LIN {X 0,Y 185.517,Z 546.376,A -85,B 0,C 180,E1 -22264.627,E2 -22264.627} C_VEL
LIN {X 0,Y 185.564,Z 546.364,A -85,B 0,C 180,E1 -22267.314,E2 -22267.314} C_VEL
LIN {X 0,Y 185.581,Z 546.361,A -85,B 0,C 180,E1 -22270.766,E2 -22270.766} C_VEL
LIN {X 0,Y 185.578,Z 546.362,A -85,B 0,C 180,E1 -22276.016,E2 -22276.016} C_VEL
LIN {X 0,Y 185.556,Z 546.364,A -85,B 0,C 180,E1 -22279.92,E2 -22279.92} C_VEL
LIN {X 0,Y 185.571,Z 546.368,A -85,B 0,C 180,E1 -22282.704,E2 -22282.704} C_VEL
LIN {X 0,Y 185.54,Z 546.354,A -85,B 0,C 180,E1 -22287.976,E2 -22287.976} C_VEL
LIN {X 0,Y 185.578,Z 546.361,A -85,B 0,C 180,E1 -22290.576,E2 -22290.576} C_VEL
LIN {X 0,Y 185.575,Z 546.366,A -85,B 0,C 180,E1 -22295.382,E2 -22295.382} C_VEL
LIN {X 0,Y 185.668,Z 546.345,A -85,B 0,C 180,E1 -22301.136,E2 -22301.136} C_VEL
LIN {X 0,Y 185.689,Z 546.352,A -85,B 0,C 180,E1 -22304.638,E2 -22304.638} C_VEL
LIN {X 0,Y 185.92,Z 546.306,A -85,B 0,C 180,E1 -22309.36,E2 -22309.36} C_VEL
LIN {X 0,Y 185.958,Z 546.315,A -85,B 0,C 180,E1 -22313.491,E2 -22313.491} C_VEL
LIN {X 0,Y 186.204,Z 546.281,A -85,B 0,C 180,E1 -22317.838,E2 -22317.838} C_VEL
LIN {X 0,Y 186.405,Z 546.247,A -85,B 0,C 180,E1 -22320.001,E2 -22320.001} C_VEL
LIN {X 0,Y 185.935,Z 546.319,A -85,B 0,C 180,E1 -22324.337,E2 -22324.337} C_VEL
LIN {X 0,Y 185.984,Z 546.307,A -85,B 0,C 180,E1 -22328.695,E2 -22328.695} C_VEL
LIN {X 0,Y 185.726,Z 546.349,A -85,B 0,C 180,E1 -22333.124,E2 -22333.124} C_VEL
LIN {X 0,Y 185.687,Z 546.346,A -85,B 0,C 180,E1 -22337.626,E2 -22337.626} C_VEL
LIN {X 0,Y 185.595,Z 546.364,A -85,B 0,C 180,E1 -22342.253,E2 -22342.253} C_VEL
LIN {X 0,Y 185.561,Z 546.372,A -85,B 0,C 180,E1 -22347.033,E2 -22347.033} C_VEL
LIN {X 0,Y 185.578,Z 546.364,A -85,B 0,C 180,E1 -22349.494,E2 -22349.494} C_VEL
LIN {X 0,Y 185.518,Z 546.372,A -85,B 0,C 180,E1 -22354.629,E2 -22354.629} C_VEL
LIN {X 0,Y 185.544,Z 546.371,A -85,B 0,C 180,E1 -22357.305,E2 -22357.305} C_VEL
LIN {X 0,Y 185.492,Z 546.377,A -85,B 0,C 180,E1 -22360.734,E2 -22360.734} C_VEL
LIN {X 0,Y 185.569,Z 546.427,A -85,B 0,C 180,E1 -22365.591,E2 -22365.591} C_VEL
LIN {X 0,Y 187.78,Z 555.622,A -85,B 0,C 180,E1 -22370.488,E2 -22370.488} C_VEL
LIN {X 0,Y 187.975,Z 556.393,A -85,B 0,C 180,E1 -22370.714,E2 -22370.714} C_VEL
LIN {X 0,Y 195.844,Z 575.592,A -85,B 0,C 180,E1 -22372.988,E2 -22372.988} C_VEL
LIN {X 0,Y 200.611,Z 588.551,A -85,B 0,C 180,E1 -22374.325,E2 -22374.325} C_VEL
LIN {X 0,Y 203.905,Z 619.674,A -85,B 0,C 180,E1 -22376.185,E2 -22376.185} C_VEL
LIN {X 0,Y 202.479,Z 649.546,A -85,B 0,C 180,E1 -22377.312,E2 -22377.312} C_VEL
LIN {X 0,Y 201.533,Z 655.365,A -85,B 0,C 180,E1 -22377.442,E2 -22377.442} C_VEL
LIN {X 0,Y 198.317,Z 664.756,A -85,B 0,C 180,E1 -22377.495,E2 -22377.495} C_VEL
LIN {X 0,Y 194.902,Z 674.04,A -85,B 0,C 180,E1 -22377.731,E2 -22377.731} C_VEL
LIN {X 0,Y 193.615,Z 679.689,A -85,B 0,C 180,E1 -22378.095,E2 -22378.095} C_VEL
LIN {X 0,Y 191.784,Z 691.638,A -85,B 0,C 180,E1 -22379.287,E2 -22379.287} C_VEL
LIN {X 0,Y 189.555,Z 703.367,A -85,B 0,C 180,E1 -22380.882,E2 -22380.882} C_VEL
LIN {X 0,Y 186.984,Z 714.728,A -85,B 0,C 180,E1 -22382.889,E2 -22382.889} C_VEL
LIN {X 0,Y 184.523,Z 725.042,A -85,B 0,C 180,E1 -22385.232,E2 -22385.232} C_VEL
LIN {X 0,Y 182.216,Z 734.209,A -85,B 0,C 180,E1 -22387.873,E2 -22387.873} C_VEL
LIN {X 0,Y 180.274,Z 741.969,A -85,B 0,C 180,E1 -22390.648,E2 -22390.648} C_VEL
LIN {X 0,Y 178.473,Z 749.457,A -85,B 0,C 180,E1 -22394,E2 -22394} C_VEL
LIN {X 0,Y 177.209,Z 755.433,A -85,B 0,C 180,E1 -22397.401,E2 -22397.401} C_VEL
LIN {X 0,Y 176.559,Z 760.116,A -85,B 0,C 180,E1 -22400.839,E2 -22400.839} C_VEL
LIN {X 0,Y 176.397,Z 764.143,A -85,B 0,C 180,E1 -22404.915,E2 -22404.915} C_VEL
LIN {X 0,Y 176.439,Z 766.075,A -85,B 0,C 180,E1 -22407.717,E2 -22407.717} C_VEL
LIN {X 0,Y 176.506,Z 767.141,A -85,B 0,C 180,E1 -22410,E2 -22410} C_VEL
LIN {X 0,Y 176.35,Z 767.745,A -85,B 0,C 180,E1 -22412.284,E2 -22412.284} C_VEL
LIN {X 0,Y 176.194,Z 767.759,A -85,B 0,C 180,E1 -22416.873,E2 -22416.873} C_VEL
LIN {X 0,Y 176.425,Z 767.177,A -85,B 0,C 180,E1 -22419.168,E2 -22419.168} C_VEL
LIN {X 0,Y 177.547,Z 764.782,A -85,B 0,C 180,E1 -22423.739,E2 -22423.739} C_VEL
LIN {X 0,Y 179.222,Z 761.932,A -85,B 0,C 180,E1 -22427.103,E2 -22427.103} C_VEL
LIN {X 0,Y 181.458,Z 758.092,A -85,B 0,C 180,E1 -22430.4,E2 -22430.4} C_VEL
LIN {X 0,Y 184.566,Z 752.928,A -85,B 0,C 180,E1 -22433.731,E2 -22433.731} C_VEL
LIN {X 0,Y 188.364,Z 745.947,A -85,B 0,C 180,E1 -22437.197,E2 -22437.197} C_VEL
LIN {X 0,Y 192.524,Z 738.16,A -85,B 0,C 180,E1 -22440.127,E2 -22440.127} C_VEL
LIN {X 0,Y 197.285,Z 728.483,A -85,B 0,C 180,E1 -22442.905,E2 -22442.905} C_VEL
LIN {X 0,Y 201.625,Z 718.591,A -85,B 0,C 180,E1 -22445.108,E2 -22445.108} C_VEL
LIN {X 0,Y 205.882,Z 707.605,A -85,B 0,C 180,E1 -22446.987,E2 -22446.987} C_VEL
LIN {X 0,Y 209.356,Z 697.038,A -85,B 0,C 180,E1 -22448.391,E2 -22448.391} C_VEL
LIN {X 0,Y 212.547,Z 685.576,A -85,B 0,C 180,E1 -22449.531,E2 -22449.531} C_VEL
LIN {X 0,Y 215.285,Z 672.899,A -85,B 0,C 180,E1 -22450.452,E2 -22450.452} C_VEL
LIN {X 0,Y 217.072,Z 659.892,A -85,B 0,C 180,E1 -22451.115,E2 -22451.115} C_VEL
LIN {X 0,Y 219.901,Z 624.876,A -85,B 0,C 180,E1 -22452.357,E2 -22452.357} C_VEL
LIN {X 0,Y 219.369,Z 614.997,A -85,B 0,C 180,E1 -22453.156,E2 -22453.156} C_VEL
LIN {X 0,Y 215.934,Z 605.716,A -85,B 0,C 180,E1 -22455.054,E2 -22455.054} C_VEL
LIN {X 0,Y 212.067,Z 596.949,A -85,B 0,C 180,E1 -22457.291,E2 -22457.291} C_VEL
LIN {X 0,Y 208.689,Z 590.362,A -85,B 0,C 180,E1 -22459.448,E2 -22459.448} C_VEL
LIN {X 0,Y 206.695,Z 586.633,A -85,B 0,C 180,E1 -22460.819,E2 -22460.819} C_VEL
LIN {X 0,Y 204.07,Z 581.906,A -85,B 0,C 180,E1 -22462.843,E2 -22462.843} C_VEL
LIN {X 0,Y 200.633,Z 575.973,A -85,B 0,C 180,E1 -22465.911,E2 -22465.911} C_VEL
LIN {X 0,Y 196.518,Z 569.368,A -85,B 0,C 180,E1 -22470.809,E2 -22470.809} C_VEL
LIN {X 0,Y 193.752,Z 565.553,A -85,B 0,C 180,E1 -22476.225,E2 -22476.225} C_VEL
LIN {X 0,Y 193.121,Z 564.144,A -85,B 0,C 180,E1 -22479.251,E2 -22479.251} C_VEL
LIN {X 0,Y 193.05,Z 563.979,A -85,B 0,C 180,E1 -22483.067,E2 -22483.067} C_VEL
LIN {X 0,Y 195.749,Z 565.397,A -85,B 0,C 180,E1 -22490.374,E2 -22490.374} C_VEL
LIN {X 0,Y 197.208,Z 568.439,A -85,B 0,C 180,E1 -22492.778,E2 -22492.778} C_VEL
LIN {X 0,Y 199.601,Z 570.637,A -85,B 0,C 180,E1 -22495.487,E2 -22495.487} C_VEL
LIN {X 0,Y 200.336,Z 571.297,A -85,B 0,C 180,E1 -22496.201,E2 -22496.201} C_VEL
LIN {X 0,Y 202.709,Z 574.7,A -85,B 0,C 180,E1 -22498.455,E2 -22498.455} C_VEL
LIN {X 0,Y 206.086,Z 579.678,A -85,B 0,C 180,E1 -22501.122,E2 -22501.122} C_VEL
LIN {X 0,Y 210.138,Z 585.674,A -85,B 0,C 180,E1 -22503.834,E2 -22503.834} C_VEL
LIN {X 0,Y 215.436,Z 594.551,A -85,B 0,C 180,E1 -22506.911,E2 -22506.911} C_VEL
LIN {X 0,Y 219.159,Z 601.544,A -85,B 0,C 180,E1 -22508.844,E2 -22508.844} C_VEL
LIN {X 0,Y 221.223,Z 605.714,A -85,B 0,C 180,E1 -22509.853,E2 -22509.853} C_VEL
LIN {X 0,Y 217.676,Z 648.267,A -85,B 0,C 180,E1 -22511.39,E2 -22511.39} C_VEL
LIN {X 0,Y 215.672,Z 661.882,A -85,B 0,C 180,E1 -22512.224,E2 -22512.224} C_VEL
LIN {X 0,Y 213.173,Z 674.111,A -85,B 0,C 180,E1 -22513.342,E2 -22513.342} C_VEL
LIN {X 0,Y 210.175,Z 685.358,A -85,B 0,C 180,E1 -22514.715,E2 -22514.715} C_VEL
LIN {X 0,Y 206.233,Z 697.154,A -85,B 0,C 180,E1 -22516.568,E2 -22516.568} C_VEL
LIN {X 0,Y 202.085,Z 707.52,A -85,B 0,C 180,E1 -22518.702,E2 -22518.702} C_VEL
LIN {X 0,Y 197.666,Z 717.189,A -85,B 0,C 180,E1 -22521.271,E2 -22521.271} C_VEL
LIN {X 0,Y 193.61,Z 724.993,A -85,B 0,C 180,E1 -22523.922,E2 -22523.922} C_VEL
LIN {X 0,Y 189.421,Z 732.125,A -85,B 0,C 180,E1 -22527.071,E2 -22527.071} C_VEL
LIN {X 0,Y 186.39,Z 736.986,A -85,B 0,C 180,E1 -22529.863,E2 -22529.863} C_VEL
LIN {X 0,Y 183.741,Z 740.865,A -85,B 0,C 180,E1 -22532.704,E2 -22532.704} C_VEL
LIN {X 0,Y 180.564,Z 745.035,A -85,B 0,C 180,E1 -22537.071,E2 -22537.071} C_VEL
LIN {X 0,Y 178.287,Z 747.512,A -85,B 0,C 180,E1 -22541.5,E2 -22541.5} C_VEL
LIN {X 0,Y 176.895,Z 748.349,A -85,B 0,C 180,E1 -22545.652,E2 -22545.652} C_VEL
LIN {X 0,Y 176.092,Z 747.755,A -85,B 0,C 180,E1 -22550.315,E2 -22550.315} C_VEL
LIN {X 0,Y 175.986,Z 746.527,A -85,B 0,C 180,E1 -22553.201,E2 -22553.201} C_VEL
LIN {X 0,Y 176.304,Z 744.071,A -85,B 0,C 180,E1 -22556.835,E2 -22556.835} C_VEL
LIN {X 0,Y 177.175,Z 740.148,A -85,B 0,C 180,E1 -22560.769,E2 -22560.769} C_VEL
LIN {X 0,Y 178.282,Z 735.346,A -85,B 0,C 180,E1 -22564.303,E2 -22564.303} C_VEL
LIN {X 0,Y 179.981,Z 728.514,A -85,B 0,C 180,E1 -22568.114,E2 -22568.114} C_VEL
LIN {X 0,Y 181.997,Z 720.884,A -85,B 0,C 180,E1 -22571.423,E2 -22571.423} C_VEL
LIN {X 0,Y 184.362,Z 711.833,A -85,B 0,C 180,E1 -22574.524,E2 -22574.524} C_VEL
LIN {X 0,Y 186.903,Z 701.354,A -85,B 0,C 180,E1 -22577.332,E2 -22577.332} C_VEL
LIN {X 0,Y 189.262,Z 690.78,A -85,B 0,C 180,E1 -22579.571,E2 -22579.571} C_VEL
LIN {X 0,Y 191.53,Z 678.663,A -85,B 0,C 180,E1 -22581.56,E2 -22581.56} C_VEL
LIN {X 0,Y 193.414,Z 666.412,A -85,B 0,C 180,E1 -22583.087,E2 -22583.087} C_VEL
LIN {X 0,Y 194.854,Z 653.682,A -85,B 0,C 180,E1 -22584.243,E2 -22584.243} C_VEL
LIN {X 0,Y 195.962,Z 639.684,A -85,B 0,C 180,E1 -22585.049,E2 -22585.049} C_VEL
LIN {X 0,Y 198.703,Z 589.027,A -85,B 0,C 180,E1 -22586.989,E2 -22586.989} C_VEL
LIN {X 0,Y 192.071,Z 573.5,A -85,B 0,C 180,E1 -22588.782,E2 -22588.782} C_VEL
LIN {X 0,Y 182.607,Z 554.067,A -85,B 0,C 180,E1 -22591.435,E2 -22591.435} C_VEL
LIN {X 0,Y 180.336,Z 550.24,A -85,B 0,C 180,E1 -22592.077,E2 -22592.077} C_VEL
LIN {X 0,Y 179.153,Z 547.494,A -85,B 0,C 180,E1 -22592.459,E2 -22592.459} C_VEL
LIN {X 0,Y 179.086,Z 547.178,A -85,B 0,C 180,E1 -22592.53,E2 -22592.53} C_VEL
LIN {X 0,Y 178.976,Z 547.189,A -85,B 0,C 180,E1 -22599.037,E2 -22599.037} C_VEL
LIN {X 0,Y 178.685,Z 547.223,A -85,B 0,C 180,E1 -22603.65,E2 -22603.65} C_VEL
LIN {X 0,Y 178.647,Z 547.229,A -85,B 0,C 180,E1 -22608.344,E2 -22608.344} C_VEL
LIN {X 0,Y 178.508,Z 547.247,A -85,B 0,C 180,E1 -22613.185,E2 -22613.185} C_VEL
LIN {X 0,Y 178.484,Z 547.251,A -85,B 0,C 180,E1 -22618.197,E2 -22618.197} C_VEL
LIN {X 0,Y 178.476,Z 547.253,A -85,B 0,C 180,E1 -22620.791,E2 -22620.791} C_VEL
LIN {X 0,Y 178.481,Z 547.251,A -85,B 0,C 180,E1 -22624.22,E2 -22624.22} C_VEL
LIN {X 0,Y 178.482,Z 547.241,A -85,B 0,C 180,E1 -22629.051,E2 -22629.051} C_VEL
LIN {X 0,Y 178.513,Z 547.246,A -85,B 0,C 180,E1 -22632.011,E2 -22632.011} C_VEL
LIN {X 0,Y 178.525,Z 547.243,A -85,B 0,C 180,E1 -22635.12,E2 -22635.12} C_VEL
LIN {X 0,Y 178.508,Z 547.232,A -85,B 0,C 180,E1 -22638.42,E2 -22638.42} C_VEL
LIN {X 0,Y 178.484,Z 547.249,A -85,B 0,C 180,E1 -22643.799,E2 -22643.799} C_VEL
LIN {X 0,Y 178.487,Z 547.24,A -85,B 0,C 180,E1 -22646.548,E2 -22646.548} C_VEL
LIN {X 0,Y 178.518,Z 547.239,A -85,B 0,C 180,E1 -22650.007,E2 -22650.007} C_VEL
LIN {X 0,Y 178.515,Z 547.248,A -85,B 0,C 180,E1 -22654.886,E2 -22654.886} C_VEL
LIN {X 0,Y 178.616,Z 547.221,A -85,B 0,C 180,E1 -22660.787,E2 -22660.787} C_VEL
LIN {X 0,Y 178.656,Z 547.227,A -85,B 0,C 180,E1 -22666.349,E2 -22666.349} C_VEL
LIN {X 0,Y 178.934,Z 547.174,A -85,B 0,C 180,E1 -22670.962,E2 -22670.962} C_VEL
LIN {X 0,Y 179.15,Z 547.16,A -85,B 0,C 180,E1 -22677.753,E2 -22677.753} C_VEL
LIN {X 0,Y 179.368,Z 547.123,A -85,B 0,C 180,E1 -22680.001,E2 -22680.001} C_VEL
LIN {X 0,Y 178.882,Z 547.198,A -85,B 0,C 180,E1 -22684.508,E2 -22684.508} C_VEL
LIN {X 0,Y 178.911,Z 547.186,A -85,B 0,C 180,E1 -22689.041,E2 -22689.041} C_VEL
LIN {X 0,Y 178.654,Z 547.23,A -85,B 0,C 180,E1 -22693.654,E2 -22693.654} C_VEL
LIN {X 0,Y 178.621,Z 547.231,A -85,B 0,C 180,E1 -22699.217,E2 -22699.217} C_VEL
LIN {X 0,Y 178.523,Z 547.242,A -85,B 0,C 180,E1 -22705.119,E2 -22705.119} C_VEL
LIN {X 0,Y 178.522,Z 547.243,A -85,B 0,C 180,E1 -22709.995,E2 -22709.995} C_VEL
LIN {X 0,Y 178.495,Z 547.247,A -85,B 0,C 180,E1 -22714.226,E2 -22714.226} C_VEL
LIN {X 0,Y 178.421,Z 547.262,A -85,B 0,C 180,E1 -22719.069,E2 -22719.069} C_VEL
LIN {X 0,Y 178.493,Z 547.298,A -85,B 0,C 180,E1 -22724.67,E2 -22724.67} C_VEL
LIN {X 0,Y 180.414,Z 555.176,A -85,B 0,C 180,E1 -22729.08,E2 -22729.08} C_VEL
LIN {X 0,Y 180.613,Z 555.846,A -85,B 0,C 180,E1 -22729.316,E2 -22729.316} C_VEL
LIN {X 0,Y 188.551,Z 574.701,A -85,B 0,C 180,E1 -22731.729,E2 -22731.729} C_VEL
LIN {X 0,Y 194.574,Z 591.255,A -85,B 0,C 180,E1 -22733.529,E2 -22733.529} C_VEL
LIN {X 0,Y 197.522,Z 620.88,A -85,B 0,C 180,E1 -22735.353,E2 -22735.353} C_VEL
LIN {X 0,Y 195.045,Z 666.296,A -85,B 0,C 180,E1 -22737.172,E2 -22737.172} C_VEL
LIN {X 0,Y 193.812,Z 678.176,A -85,B 0,C 180,E1 -22737.973,E2 -22737.973} C_VEL
LIN {X 0,Y 193.615,Z 679.689,A -85,B 0,C 180,E1 -22738.095,E2 -22738.095} C_VEL
LIN {X 0,Y 192.148,Z 685.25,A -85,B 0,C 180,E1 -22738.513,E2 -22738.513} C_VEL
LIN {X 0,Y 187.941,Z 694.002,A -85,B 0,C 180,E1 -22739.154,E2 -22739.154} C_VEL
LIN {X 0,Y 183.605,Z 702.435,A -85,B 0,C 180,E1 -22740.042,E2 -22740.042} C_VEL
LIN {X 0,Y 181.958,Z 707.489,A -85,B 0,C 180,E1 -22740.843,E2 -22740.843} C_VEL
LIN {X 0,Y 179.215,Z 719.04,A -85,B 0,C 180,E1 -22743.194,E2 -22743.194} C_VEL
LIN {X 0,Y 177.031,Z 727.49,A -85,B 0,C 180,E1 -22745.365,E2 -22745.365} C_VEL
LIN {X 0,Y 174.552,Z 736.495,A -85,B 0,C 180,E1 -22748.221,E2 -22748.221} C_VEL
LIN {X 0,Y 172.508,Z 744.812,A -85,B 0,C 180,E1 -22751.595,E2 -22751.595} C_VEL
LIN {X 0,Y 170.822,Z 751.631,A -85,B 0,C 180,E1 -22755.1,E2 -22755.1} C_VEL
LIN {X 0,Y 169.697,Z 757.854,A -85,B 0,C 180,E1 -22759.259,E2 -22759.259} C_VEL
LIN {X 0,Y 169.31,Z 761.846,A -85,B 0,C 180,E1 -22762.847,E2 -22762.847} C_VEL
LIN {X 0,Y 169.328,Z 763.874,A -85,B 0,C 180,E1 -22765.238,E2 -22765.238} C_VEL
LIN {X 0,Y 169.355,Z 765.452,A -85,B 0,C 180,E1 -22767.622,E2 -22767.622} C_VEL
LIN {X 0,Y 169.44,Z 766.598,A -85,B 0,C 180,E1 -22770,E2 -22770} C_VEL
LIN {X 0,Y 169.114,Z 767.495,A -85,B 0,C 180,E1 -22774.131,E2 -22774.131} C_VEL
LIN {X 0,Y 169.126,Z 767.366,A -85,B 0,C 180,E1 -22777.161,E2 -22777.161} C_VEL
LIN {X 0,Y 169.379,Z 766.846,A -85,B 0,C 180,E1 -22779.553,E2 -22779.553} C_VEL
LIN {X 0,Y 169.863,Z 765.923,A -85,B 0,C 180,E1 -22781.939,E2 -22781.939} C_VEL
LIN {X 0,Y 171.721,Z 762.851,A -85,B 0,C 180,E1 -22786.647,E2 -22786.647} C_VEL
LIN {X 0,Y 173.974,Z 759.469,A -85,B 0,C 180,E1 -22790.082,E2 -22790.082} C_VEL
LIN {X 0,Y 176.85,Z 755.059,A -85,B 0,C 180,E1 -22793.415,E2 -22793.415} C_VEL
LIN {X 0,Y 180.784,Z 748.483,A -85,B 0,C 180,E1 -22797.179,E2 -22797.179} C_VEL
LIN {X 0,Y 184.954,Z 741.38,A -85,B 0,C 180,E1 -22800.23,E2 -22800.23} C_VEL
LIN {X 0,Y 189.674,Z 732.613,A -85,B 0,C 180,E1 -22803.129,E2 -22803.129} C_VEL
LIN {X 0,Y 194.104,Z 723.731,A -85,B 0,C 180,E1 -22805.402,E2 -22805.402} C_VEL
LIN {X 0,Y 198.793,Z 712.911,A -85,B 0,C 180,E1 -22807.577,E2 -22807.577} C_VEL
LIN {X 0,Y 202.843,Z 702.103,A -85,B 0,C 180,E1 -22809.22,E2 -22809.22} C_VEL
LIN {X 0,Y 206.595,Z 690.184,A -85,B 0,C 180,E1 -22810.585,E2 -22810.585} C_VEL
LIN {X 0,Y 209.73,Z 677.93,A -85,B 0,C 180,E1 -22811.598,E2 -22811.598} C_VEL
LIN {X 0,Y 212.106,Z 664.304,A -85,B 0,C 180,E1 -22812.4,E2 -22812.4} C_VEL
LIN {X 0,Y 214.091,Z 644.025,A -85,B 0,C 180,E1 -22813.158,E2 -22813.158} C_VEL
LIN {X 0,Y 215.57,Z 625.879,A -85,B 0,C 180,E1 -22813.819,E2 -22813.819} C_VEL
LIN {X 0,Y 215.277,Z 618.3,A -85,B 0,C 180,E1 -22814.445,E2 -22814.445} C_VEL
LIN {X 0,Y 211.9,Z 609.02,A -85,B 0,C 180,E1 -22816.466,E2 -22816.466} C_VEL
LIN {X 0,Y 208.766,Z 601.726,A -85,B 0,C 180,E1 -22818.464,E2 -22818.464} C_VEL
LIN {X 0,Y 205.691,Z 595.44,A -85,B 0,C 180,E1 -22820.575,E2 -22820.575} C_VEL
LIN {X 0,Y 203.613,Z 591.42,A -85,B 0,C 180,E1 -22822.167,E2 -22822.167} C_VEL
LIN {X 0,Y 201.707,Z 587.854,A -85,B 0,C 180,E1 -22823.759,E2 -22823.759} C_VEL
LIN {X 0,Y 198.706,Z 582.299,A -85,B 0,C 180,E1 -22826.677,E2 -22826.677} C_VEL
LIN {X 0,Y 195.087,Z 576.109,A -85,B 0,C 180,E1 -22831.317,E2 -22831.317} C_VEL
LIN {X 0,Y 192.499,Z 572.282,A -85,B 0,C 180,E1 -22836.89,E2 -22836.89} C_VEL
LIN {X 0,Y 192.023,Z 571.108,A -85,B 0,C 180,E1 -22839.722,E2 -22839.722} C_VEL
LIN {X 0,Y 192.16,Z 571.117,A -85,B 0,C 180,E1 -22844.079,E2 -22844.079} C_VEL
LIN {X 0,Y 194.484,Z 572.512,A -85,B 0,C 180,E1 -22850.099,E2 -22850.099} C_VEL
LIN {X 0,Y 196.01,Z 575.569,A -85,B 0,C 180,E1 -22852.652,E2 -22852.652} C_VEL
LIN {X 0,Y 198.624,Z 577.973,A -85,B 0,C 180,E1 -22855.631,E2 -22855.631} C_VEL
LIN {X 0,Y 201.392,Z 582.172,A -85,B 0,C 180,E1 -22858.366,E2 -22858.366} C_VEL
LIN {X 0,Y 204.038,Z 586.131,A -85,B 0,C 180,E1 -22860.514,E2 -22860.514} C_VEL
LIN {X 0,Y 207.661,Z 591.827,A -85,B 0,C 180,E1 -22863.105,E2 -22863.105} C_VEL
LIN {X 0,Y 212.638,Z 600.542,A -85,B 0,C 180,E1 -22866.18,E2 -22866.18} C_VEL
LIN {X 0,Y 216.291,Z 607.643,A -85,B 0,C 180,E1 -22868.166,E2 -22868.166} C_VEL
LIN {X 0,Y 216.856,Z 608.973,A -85,B 0,C 180,E1 -22868.474,E2 -22868.474} C_VEL
LIN {X 0,Y 213.287,Z 648.802,A -85,B 0,C 180,E1 -22869.918,E2 -22869.918} C_VEL
LIN {X 0,Y 211.178,Z 662.261,A -85,B 0,C 180,E1 -22870.741,E2 -22870.741} C_VEL
LIN {X 0,Y 208.758,Z 673.849,A -85,B 0,C 180,E1 -22871.804,E2 -22871.804} C_VEL
LIN {X 0,Y 205.462,Z 685.712,A -85,B 0,C 180,E1 -22873.243,E2 -22873.243} C_VEL
LIN {X 0,Y 201.804,Z 696.255,A -85,B 0,C 180,E1 -22874.882,E2 -22874.882} C_VEL
LIN {X 0,Y 197.506,Z 706.815,A -85,B 0,C 180,E1 -22877.004,E2 -22877.004} C_VEL
LIN {X 0,Y 192.914,Z 716.379,A -85,B 0,C 180,E1 -22879.504,E2 -22879.504} C_VEL
LIN {X 0,Y 188.173,Z 725.092,A -85,B 0,C 180,E1 -22882.463,E2 -22882.463} C_VEL
LIN {X 0,Y 183.333,Z 732.845,A -85,B 0,C 180,E1 -22885.959,E2 -22885.959} C_VEL
LIN {X 0,Y 179.994,Z 737.794,A -85,B 0,C 180,E1 -22888.919,E2 -22888.919} C_VEL
LIN {X 0,Y 176.169,Z 742.919,A -85,B 0,C 180,E1 -22893.098,E2 -22893.098} C_VEL
LIN {X 0,Y 173.118,Z 746.408,A -85,B 0,C 180,E1 -22897.512,E2 -22897.512} C_VEL
LIN {X 0,Y 170.85,Z 748.399,A -85,B 0,C 180,E1 -22902.233,E2 -22902.233} C_VEL
LIN {X 0,Y 169.894,Z 748.785,A -85,B 0,C 180,E1 -22905.314,E2 -22905.314} C_VEL
LIN {X 0,Y 169.252,Z 748.551,A -85,B 0,C 180,E1 -22908.366,E2 -22908.366} C_VEL
LIN {X 0,Y 168.89,Z 747.283,A -85,B 0,C 180,E1 -22912.244,E2 -22912.244} C_VEL
LIN {X 0,Y 169.106,Z 744.855,A -85,B 0,C 180,E1 -22916.219,E2 -22916.219} C_VEL
LIN {X 0,Y 169.946,Z 741.111,A -85,B 0,C 180,E1 -22920.276,E2 -22920.276} C_VEL
LIN {X 0,Y 171.241,Z 735.638,A -85,B 0,C 180,E1 -22924.541,E2 -22924.541} C_VEL
LIN {X 0,Y 173.034,Z 728.659,A -85,B 0,C 180,E1 -22928.559,E2 -22928.559} C_VEL
LIN {X 0,Y 175.02,Z 721.458,A -85,B 0,C 180,E1 -22931.798,E2 -22931.798} C_VEL
LIN {X 0,Y 177.5,Z 712.235,A -85,B 0,C 180,E1 -22935.087,E2 -22935.087} C_VEL
LIN {X 0,Y 180.135,Z 701.766,A -85,B 0,C 180,E1 -22937.993,E2 -22937.993} C_VEL
LIN {X 0,Y 182.583,Z 691.199,A -85,B 0,C 180,E1 -22940.305,E2 -22940.305} C_VEL
LIN {X 0,Y 184.939,Z 679.122,A -85,B 0,C 180,E1 -22942.353,E2 -22942.353} C_VEL
LIN {X 0,Y 186.915,Z 666.847,A -85,B 0,C 180,E1 -22943.93,E2 -22943.93} C_VEL
LIN {X 0,Y 188.406,Z 654.178,A -85,B 0,C 180,E1 -22945.119,E2 -22945.119} C_VEL
LIN {X 0,Y 189.579,Z 639.972,A -85,B 0,C 180,E1 -22945.962,E2 -22945.962} C_VEL
LIN {X 0,Y 192.341,Z 590.76,A -85,B 0,C 180,E1 -22947.906,E2 -22947.906} C_VEL
LIN {X 0,Y 186.259,Z 576.62,A -85,B 0,C 180,E1 -22949.607,E2 -22949.607} C_VEL
LIN {X 0,Y 177.456,Z 558.29,A -85,B 0,C 180,E1 -22952.217,E2 -22952.217} C_VEL
LIN {X 0,Y 173.599,Z 551.821,A -85,B 0,C 180,E1 -22953.361,E2 -22953.361} C_VEL
LIN {X 0,Y 172.119,Z 549.158,A -85,B 0,C 180,E1 -22953.826,E2 -22953.826} C_VEL
LIN {X 0,Y 171.865,Z 548.078,A -85,B 0,C 180,E1 -22954.03,E2 -22954.03} C_VEL
LIN {X 0,Y 171.908,Z 548.07,A -85,B 0,C 180,E1 -22959.412,E2 -22959.412} C_VEL
LIN {X 0,Y 171.607,Z 548.104,A -85,B 0,C 180,E1 -22964.224,E2 -22964.224} C_VEL
LIN {X 0,Y 171.541,Z 548.112,A -85,B 0,C 180,E1 -22969.562,E2 -22969.562} C_VEL
LIN {X 0,Y 171.466,Z 548.122,A -85,B 0,C 180,E1 -22975.616,E2 -22975.616} C_VEL
LIN {X 0,Y 171.438,Z 548.128,A -85,B 0,C 180,E1 -22980.587,E2 -22980.587} C_VEL
LIN {X 0,Y 171.436,Z 548.132,A -85,B 0,C 180,E1 -22985.024,E2 -22985.024} C_VEL
LIN {X 0,Y 171.435,Z 548.118,A -85,B 0,C 180,E1 -22988.841,E2 -22988.841} C_VEL
LIN {X 0,Y 171.449,Z 548.127,A -85,B 0,C 180,E1 -22994.174,E2 -22994.174} C_VEL
LIN {X 0,Y 171.425,Z 548.116,A -85,B 0,C 180,E1 -22999.009,E2 -22999.009} C_VEL
LIN {X 0,Y 171.438,Z 548.127,A -85,B 0,C 180,E1 -23002.056,E2 -23002.056} C_VEL
LIN {X 0,Y 171.412,Z 548.127,A -85,B 0,C 180,E1 -23005.084,E2 -23005.084} C_VEL
LIN {X 0,Y 171.444,Z 548.12,A -85,B 0,C 180,E1 -23010.535,E2 -23010.535} C_VEL
LIN {X 0,Y 171.44,Z 548.125,A -85,B 0,C 180,E1 -23015.8,E2 -23015.8} C_VEL
LIN {X 0,Y 171.572,Z 548.098,A -85,B 0,C 180,E1 -23020.872,E2 -23020.872} C_VEL
LIN {X 0,Y 171.573,Z 548.11,A -85,B 0,C 180,E1 -23025.774,E2 -23025.774} C_VEL
LIN {X 0,Y 171.869,Z 548.052,A -85,B 0,C 180,E1 -23030.587,E2 -23030.587} C_VEL
LIN {X 0,Y 171.82,Z 548.079,A -85,B 0,C 180,E1 -23035.309,E2 -23035.309} C_VEL
LIN {X 0,Y 172.331,Z 547.999,A -85,B 0,C 180,E1 -23040.001,E2 -23040.001} C_VEL
LIN {X 0,Y 171.829,Z 548.077,A -85,B 0,C 180,E1 -23044.693,E2 -23044.693} C_VEL
LIN {X 0,Y 171.847,Z 548.064,A -85,B 0,C 180,E1 -23049.416,E2 -23049.416} C_VEL
LIN {X 0,Y 171.573,Z 548.111,A -85,B 0,C 180,E1 -23054.229,E2 -23054.229} C_VEL
LIN {X 0,Y 171.543,Z 548.115,A -85,B 0,C 180,E1 -23059.563,E2 -23059.563} C_VEL
LIN {X 0,Y 171.461,Z 548.125,A -85,B 0,C 180,E1 -23065.613,E2 -23065.613} C_VEL
LIN {X 0,Y 171.441,Z 548.127,A -85,B 0,C 180,E1 -23070.588,E2 -23070.588} C_VEL
LIN {X 0,Y 171.406,Z 548.132,A -85,B 0,C 180,E1 -23075.033,E2 -23075.033} C_VEL
LIN {X 0,Y 171.382,Z 548.138,A -85,B 0,C 180,E1 -23078.819,E2 -23078.819} C_VEL
LIN {X 0,Y 171.433,Z 548.18,A -85,B 0,C 180,E1 -23083.686,E2 -23083.686} C_VEL
LIN {X 0,Y 173.204,Z 555.248,A -85,B 0,C 180,E1 -23087.799,E2 -23087.799} C_VEL
LIN {X 0,Y 180.811,Z 572.906,A -85,B 0,C 180,E1 -23090.255,E2 -23090.255} C_VEL
LIN {X 0,Y 187.846,Z 591.474,A -85,B 0,C 180,E1 -23092.44,E2 -23092.44} C_VEL
LIN {X 0,Y 188.569,Z 594.359,A -85,B 0,C 180,E1 -23092.703,E2 -23092.703} C_VEL
LIN {X 0,Y 191.147,Z 620.798,A -85,B 0,C 180,E1 -23094.401,E2 -23094.401} C_VEL
LIN {X 0,Y 188.626,Z 665.85,A -85,B 0,C 180,E1 -23096.263,E2 -23096.263} C_VEL
LIN {X 0,Y 187.303,Z 678.136,A -85,B 0,C 180,E1 -23097.12,E2 -23097.12} C_VEL
LIN {X 0,Y 185.289,Z 690.967,A -85,B 0,C 180,E1 -23098.406,E2 -23098.406} C_VEL
LIN {X 0,Y 182.988,Z 702.761,A -85,B 0,C 180,E1 -23100.048,E2 -23100.048} C_VEL
LIN {X 0,Y 181.958,Z 707.489,A -85,B 0,C 180,E1 -23100.843,E2 -23100.843} C_VEL
LIN {X 0,Y 180.251,Z 712.513,A -85,B 0,C 180,E1 -23101.73,E2 -23101.73} C_VEL
LIN {X 0,Y 175.559,Z 720.135,A -85,B 0,C 180,E1 -23103.141,E2 -23103.141} C_VEL
LIN {X 0,Y 170.831,Z 727.218,A -85,B 0,C 180,E1 -23104.802,E2 -23104.802} C_VEL
LIN {X 0,Y 169.094,Z 731.386,A -85,B 0,C 180,E1 -23106.052,E2 -23106.052} C_VEL
LIN {X 0,Y 166.834,Z 739.508,A -85,B 0,C 180,E1 -23109.019,E2 -23109.019} C_VEL
LIN {X 0,Y 164.827,Z 747.311,A -85,B 0,C 180,E1 -23112.635,E2 -23112.635} C_VEL
LIN {X 0,Y 163.282,Z 753.526,A -85,B 0,C 180,E1 -23116.307,E2 -23116.307} C_VEL
LIN {X 0,Y 162.506,Z 758.444,A -85,B 0,C 180,E1 -23120.039,E2 -23120.039} C_VEL
LIN {X 0,Y 162.22,Z 762.173,A -85,B 0,C 180,E1 -23123.782,E2 -23123.782} C_VEL
LIN {X 0,Y 162.273,Z 764.815,A -85,B 0,C 180,E1 -23127.518,E2 -23127.518} C_VEL
LIN {X 0,Y 162.374,Z 766.015,A -85,B 0,C 180,E1 -23130,E2 -23130} C_VEL
LIN {X 0,Y 162.056,Z 766.997,A -85,B 0,C 180,E1 -23134.071,E2 -23134.071} C_VEL
LIN {X 0,Y 162.064,Z 766.973,A -85,B 0,C 180,E1 -23137.475,E2 -23137.475} C_VEL
LIN {X 0,Y 162.874,Z 765.654,A -85,B 0,C 180,E1 -23142.459,E2 -23142.459} C_VEL
LIN {X 0,Y 163.698,Z 764.401,A -85,B 0,C 180,E1 -23144.927,E2 -23144.927} C_VEL
LIN {X 0,Y 166.453,Z 760.658,A -85,B 0,C 180,E1 -23149.741,E2 -23149.741} C_VEL
LIN {X 0,Y 169.249,Z 756.713,A -85,B 0,C 180,E1 -23153.233,E2 -23153.233} C_VEL
LIN {X 0,Y 172.583,Z 751.692,A -85,B 0,C 180,E1 -23156.611,E2 -23156.611} C_VEL
LIN {X 0,Y 176.6,Z 745.48,A -85,B 0,C 180,E1 -23159.831,E2 -23159.831} C_VEL
LIN {X 0,Y 181.293,Z 737.837,A -85,B 0,C 180,E1 -23162.868,E2 -23162.868} C_VEL
LIN {X 0,Y 185.622,Z 730.101,A -85,B 0,C 180,E1 -23165.267,E2 -23165.267} C_VEL
LIN {X 0,Y 190.774,Z 719.712,A -85,B 0,C 180,E1 -23167.766,E2 -23167.766} C_VEL
LIN {X 0,Y 195.396,Z 709.23,A -85,B 0,C 180,E1 -23169.674,E2 -23169.674} C_VEL
LIN {X 0,Y 199.675,Z 697.747,A -85,B 0,C 180,E1 -23171.295,E2 -23171.295} C_VEL
LIN {X 0,Y 203.406,Z 685.688,A -85,B 0,C 180,E1 -23172.524,E2 -23172.524} C_VEL
LIN {X 0,Y 206.535,Z 672.446,A -85,B 0,C 180,E1 -23173.503,E2 -23173.503} C_VEL
LIN {X 0,Y 208.47,Z 659.988,A -85,B 0,C 180,E1 -23174.16,E2 -23174.16} C_VEL
LIN {X 0,Y 211.453,Z 626.855,A -85,B 0,C 180,E1 -23175.361,E2 -23175.361} C_VEL
LIN {X 0,Y 211.246,Z 621.418,A -85,B 0,C 180,E1 -23175.838,E2 -23175.838} C_VEL
LIN {X 0,Y 207.858,Z 611.861,A -85,B 0,C 180,E1 -23178.078,E2 -23178.078} C_VEL
LIN {X 0,Y 204.384,Z 603.729,A -85,B 0,C 180,E1 -23180.541,E2 -23180.541} C_VEL
LIN {X 0,Y 201.594,Z 597.976,A -85,B 0,C 180,E1 -23182.768,E2 -23182.768} C_VEL
LIN {X 0,Y 199.529,Z 593.959,A -85,B 0,C 180,E1 -23184.585,E2 -23184.585} C_VEL
LIN {X 0,Y 196.777,Z 588.577,A -85,B 0,C 180,E1 -23187.498,E2 -23187.498} C_VEL
LIN {X 0,Y 193.654,Z 582.822,A -85,B 0,C 180,E1 -23191.848,E2 -23191.848} C_VEL
LIN {X 0,Y 191.272,Z 578.98,A -85,B 0,C 180,E1 -23197.59,E2 -23197.59} C_VEL
LIN {X 0,Y 190.992,Z 578.159,A -85,B 0,C 180,E1 -23199.608,E2 -23199.608} C_VEL
LIN {X 0,Y 191.102,Z 578.113,A -85,B 0,C 180,E1 -23203.988,E2 -23203.988} C_VEL
LIN {X 0,Y 193.154,Z 579.37,A -85,B 0,C 180,E1 -23209.618,E2 -23209.618} C_VEL
LIN {X 0,Y 194.876,Z 582.735,A -85,B 0,C 180,E1 -23212.609,E2 -23212.609} C_VEL
LIN {X 0,Y 196.996,Z 584.759,A -85,B 0,C 180,E1 -23215.128,E2 -23215.128} C_VEL
LIN {X 0,Y 199.508,Z 588.702,A -85,B 0,C 180,E1 -23217.726,E2 -23217.726} C_VEL
LIN {X 0,Y 202.95,Z 594.201,A -85,B 0,C 180,E1 -23220.651,E2 -23220.651} C_VEL
LIN {X 0,Y 205.889,Z 599.007,A -85,B 0,C 180,E1 -23222.806,E2 -23222.806} C_VEL
LIN {X 0,Y 211.017,Z 608.654,A -85,B 0,C 180,E1 -23226.083,E2 -23226.083} C_VEL
LIN {X 0,Y 212.61,Z 612.105,A -85,B 0,C 180,E1 -23227.009,E2 -23227.009} C_VEL
LIN {X 0,Y 209.129,Z 649.221,A -85,B 0,C 180,E1 -23228.36,E2 -23228.36} C_VEL
LIN {X 0,Y 206.829,Z 663.322,A -85,B 0,C 180,E1 -23229.235,E2 -23229.235} C_VEL
LIN {X 0,Y 203.993,Z 675.781,A -85,B 0,C 180,E1 -23230.42,E2 -23230.42} C_VEL
LIN {X 0,Y 200.365,Z 687.816,A -85,B 0,C 180,E1 -23231.937,E2 -23231.937} C_VEL
LIN {X 0,Y 196.236,Z 698.786,A -85,B 0,C 180,E1 -23233.729,E2 -23233.729} C_VEL
LIN {X 0,Y 191.783,Z 708.795,A -85,B 0,C 180,E1 -23235.862,E2 -23235.862} C_VEL
LIN {X 0,Y 186.981,Z 718.187,A -85,B 0,C 180,E1 -23238.439,E2 -23238.439} C_VEL
LIN {X 0,Y 182.539,Z 725.818,A -85,B 0,C 180,E1 -23241.13,E2 -23241.13} C_VEL
LIN {X 0,Y 177.666,Z 733.155,A -85,B 0,C 180,E1 -23244.523,E2 -23244.523} C_VEL
LIN {X 0,Y 173.091,Z 739.391,A -85,B 0,C 180,E1 -23248.469,E2 -23248.469} C_VEL
LIN {X 0,Y 169.242,Z 744.027,A -85,B 0,C 180,E1 -23252.672,E2 -23252.672} C_VEL
LIN {X 0,Y 166.436,Z 746.929,A -85,B 0,C 180,E1 -23256.651,E2 -23256.651} C_VEL
LIN {X 0,Y 164.749,Z 748.389,A -85,B 0,C 180,E1 -23259.84,E2 -23259.84} C_VEL
LIN {X 0,Y 163.288,Z 749.182,A -85,B 0,C 180,E1 -23263.521,E2 -23263.521} C_VEL
LIN {X 0,Y 162.304,Z 749.05,A -85,B 0,C 180,E1 -23267.401,E2 -23267.401} C_VEL
LIN {X 0,Y 161.829,Z 747.908,A -85,B 0,C 180,E1 -23271.415,E2 -23271.415} C_VEL
LIN {X 0,Y 161.939,Z 745.559,A -85,B 0,C 180,E1 -23275.655,E2 -23275.655} C_VEL
LIN {X 0,Y 162.706,Z 742.06,A -85,B 0,C 180,E1 -23279.754,E2 -23279.754} C_VEL
LIN {X 0,Y 163.95,Z 736.776,A -85,B 0,C 180,E1 -23284.182,E2 -23284.182} C_VEL
LIN {X 0,Y 165.641,Z 730.382,A -85,B 0,C 180,E1 -23288.206,E2 -23288.206} C_VEL
LIN {X 0,Y 167.687,Z 723.241,A -85,B 0,C 180,E1 -23291.68,E2 -23291.68} C_VEL
LIN {X 0,Y 170.102,Z 714.539,A -85,B 0,C 180,E1 -23295.035,E2 -23295.035} C_VEL
LIN {X 0,Y 172.542,Z 705.42,A -85,B 0,C 180,E1 -23297.837,E2 -23297.837} C_VEL
LIN {X 0,Y 175.23,Z 694.495,A -85,B 0,C 180,E1 -23300.477,E2 -23300.477} C_VEL
LIN {X 0,Y 177.839,Z 682.344,A -85,B 0,C 180,E1 -23302.75,E2 -23302.75} C_VEL
LIN {X 0,Y 179.872,Z 670.841,A -85,B 0,C 180,E1 -23304.395,E2 -23304.395} C_VEL
LIN {X 0,Y 181.762,Z 657.066,A -85,B 0,C 180,E1 -23305.82,E2 -23305.82} C_VEL
LIN {X 0,Y 182.928,Z 644.837,A -85,B 0,C 180,E1 -23306.682,E2 -23306.682} C_VEL
LIN {X 0,Y 186.091,Z 592.769,A -85,B 0,C 180,E1 -23308.822,E2 -23308.822} C_VEL
LIN {X 0,Y 180.767,Z 580.362,A -85,B 0,C 180,E1 -23310.4,E2 -23310.4} C_VEL
LIN {X 0,Y 172.214,Z 562.377,A -85,B 0,C 180,E1 -23313.057,E2 -23313.057} C_VEL
LIN {X 0,Y 166.355,Z 552.606,A -85,B 0,C 180,E1 -23314.909,E2 -23314.909} C_VEL
LIN {X 0,Y 164.985,Z 550.013,A -85,B 0,C 180,E1 -23315.385,E2 -23315.385} C_VEL
LIN {X 0,Y 164.798,Z 548.958,A -85,B 0,C 180,E1 -23315.506,E2 -23315.506} C_VEL
LIN {X 0,Y 164.85,Z 548.949,A -85,B 0,C 180,E1 -23319.818,E2 -23319.818} C_VEL
LIN {X 0,Y 164.55,Z 548.985,A -85,B 0,C 180,E1 -23324.848,E2 -23324.848} C_VEL
LIN {X 0,Y 164.47,Z 548.993,A -85,B 0,C 180,E1 -23329.989,E2 -23329.989} C_VEL
LIN {X 0,Y 164.39,Z 549.003,A -85,B 0,C 180,E1 -23336.134,E2 -23336.134} C_VEL
LIN {X 0,Y 164.372,Z 549.011,A -85,B 0,C 180,E1 -23341.228,E2 -23341.228} C_VEL
LIN {X 0,Y 164.358,Z 549.008,A -85,B 0,C 180,E1 -23346.772,E2 -23346.772} C_VEL
LIN {X 0,Y 164.372,Z 548.999,A -85,B 0,C 180,E1 -23349.891,E2 -23349.891} C_VEL
LIN {X 0,Y 164.388,Z 549.008,A -85,B 0,C 180,E1 -23353.384,E2 -23353.384} C_VEL
LIN {X 0,Y 164.389,Z 548.993,A -85,B 0,C 180,E1 -23356.842,E2 -23356.842} C_VEL
LIN {X 0,Y 164.371,Z 549.003,A -85,B 0,C 180,E1 -23360.318,E2 -23360.318} C_VEL
LIN {X 0,Y 164.349,Z 549.01,A -85,B 0,C 180,E1 -23364.338,E2 -23364.338} C_VEL
LIN {X 0,Y 164.387,Z 548.99,A -85,B 0,C 180,E1 -23369.135,E2 -23369.135} C_VEL
LIN {X 0,Y 164.402,Z 549.006,A -85,B 0,C 180,E1 -23374.693,E2 -23374.693} C_VEL
LIN {X 0,Y 164.48,Z 548.977,A -85,B 0,C 180,E1 -23380.052,E2 -23380.052} C_VEL
LIN {X 0,Y 164.52,Z 548.991,A -85,B 0,C 180,E1 -23385.15,E2 -23385.15} C_VEL
LIN {X 0,Y 164.793,Z 548.932,A -85,B 0,C 180,E1 -23390.179,E2 -23390.179} C_VEL
LIN {X 0,Y 164.843,Z 548.939,A -85,B 0,C 180,E1 -23392.653,E2 -23392.653} C_VEL
LIN {X 0,Y 165.047,Z 548.917,A -85,B 0,C 180,E1 -23397.561,E2 -23397.561} C_VEL
LIN {X 0,Y 165.293,Z 548.874,A -85,B 0,C 180,E1 -23400.001,E2 -23400.001} C_VEL
LIN {X 0,Y 164.777,Z 548.956,A -85,B 0,C 180,E1 -23404.895,E2 -23404.895} C_VEL
LIN {X 0,Y 164.833,Z 548.945,A -85,B 0,C 180,E1 -23407.35,E2 -23407.35} C_VEL
LIN {X 0,Y 164.701,Z 548.959,A -85,B 0,C 180,E1 -23411.063,E2 -23411.063} C_VEL
LIN {X 0,Y 164.48,Z 548.986,A -85,B 0,C 180,E1 -23417.405,E2 -23417.405} C_VEL
LIN {X 0,Y 164.472,Z 548.997,A -85,B 0,C 180,E1 -23419.991,E2 -23419.991} C_VEL
LIN {X 0,Y 164.387,Z 549.008,A -85,B 0,C 180,E1 -23426.132,E2 -23426.132} C_VEL
LIN {X 0,Y 164.375,Z 549.009,A -85,B 0,C 180,E1 -23431.23,E2 -23431.23} C_VEL
LIN {X 0,Y 164.313,Z 549.016,A -85,B 0,C 180,E1 -23436.786,E2 -23436.786} C_VEL
LIN {X 0,Y 164.373,Z 549.082,A -85,B 0,C 180,E1 -23442.644,E2 -23442.644} C_VEL
LIN {X 0,Y 165.778,Z 554.646,A -85,B 0,C 180,E1 -23446.114,E2 -23446.114} C_VEL
LIN {X 0,Y 173.434,Z 571.944,A -85,B 0,C 180,E1 -23448.772,E2 -23448.772} C_VEL
LIN {X 0,Y 180.554,Z 590.336,A -85,B 0,C 180,E1 -23451.124,E2 -23451.124} C_VEL
LIN {X 0,Y 182.418,Z 596.012,A -85,B 0,C 180,E1 -23451.75,E2 -23451.75} C_VEL
LIN {X 0,Y 184.79,Z 622.423,A -85,B 0,C 180,E1 -23453.483,E2 -23453.483} C_VEL
LIN {X 0,Y 182.318,Z 664.617,A -85,B 0,C 180,E1 -23455.265,E2 -23455.265} C_VEL
LIN {X 0,Y 180.954,Z 677.144,A -85,B 0,C 180,E1 -23456.146,E2 -23456.146} C_VEL
LIN {X 0,Y 178.85,Z 690.101,A -85,B 0,C 180,E1 -23457.463,E2 -23457.463} C_VEL
LIN {X 0,Y 176.476,Z 702.015,A -85,B 0,C 180,E1 -23459.155,E2 -23459.155} C_VEL
LIN {X 0,Y 173.745,Z 713.472,A -85,B 0,C 180,E1 -23461.293,E2 -23461.293} C_VEL
LIN {X 0,Y 171.092,Z 723.875,A -85,B 0,C 180,E1 -23463.796,E2 -23463.796} C_VEL
LIN {X 0,Y 169.094,Z 731.386,A -85,B 0,C 180,E1 -23466.052,E2 -23466.052} C_VEL
LIN {X 0,Y 167.431,Z 735.45,A -85,B 0,C 180,E1 -23467.396,E2 -23467.396} C_VEL
LIN {X 0,Y 162.977,Z 741.472,A -85,B 0,C 180,E1 -23469.649,E2 -23469.649} C_VEL
LIN {X 0,Y 158.558,Z 746.832,A -85,B 0,C 180,E1 -23472.196,E2 -23472.196} C_VEL
LIN {X 0,Y 157.001,Z 749.868,A -85,B 0,C 180,E1 -23473.963,E2 -23473.963} C_VEL
LIN {X 0,Y 155.72,Z 756.045,A -85,B 0,C 180,E1 -23478.282,E2 -23478.282} C_VEL
LIN {X 0,Y 155.189,Z 760.274,A -85,B 0,C 180,E1 -23482.192,E2 -23482.192} C_VEL
LIN {X 0,Y 155.185,Z 762.702,A -85,B 0,C 180,E1 -23485.104,E2 -23485.104} C_VEL
LIN {X 0,Y 155.194,Z 764.179,A -85,B 0,C 180,E1 -23487.405,E2 -23487.405} C_VEL
LIN {X 0,Y 155.309,Z 765.43,A -85,B 0,C 180,E1 -23490,E2 -23490} C_VEL
LIN {X 0,Y 154.998,Z 766.472,A -85,B 0,C 180,E1 -23494.009,E2 -23494.009} C_VEL
LIN {X 0,Y 154.992,Z 766.581,A -85,B 0,C 180,E1 -23497.818,E2 -23497.818} C_VEL
LIN {X 0,Y 155.91,Z 765.37,A -85,B 0,C 180,E1 -23503.025,E2 -23503.025} C_VEL
LIN {X 0,Y 156.809,Z 764.199,A -85,B 0,C 180,E1 -23505.599,E2 -23505.599} C_VEL
LIN {X 0,Y 158.902,Z 761.656,A -85,B 0,C 180,E1 -23509.372,E2 -23509.372} C_VEL
LIN {X 0,Y 161.629,Z 758.177,A -85,B 0,C 180,E1 -23513.037,E2 -23513.037} C_VEL
LIN {X 0,Y 165.042,Z 753.644,A -85,B 0,C 180,E1 -23516.586,E2 -23516.586} C_VEL
LIN {X 0,Y 168.981,Z 748.041,A -85,B 0,C 180,E1 -23519.939,E2 -23519.939} C_VEL
LIN {X 0,Y 173.692,Z 741.081,A -85,B 0,C 180,E1 -23523.109,E2 -23523.109} C_VEL
LIN {X 0,Y 179.004,Z 732.484,A -85,B 0,C 180,E1 -23526.08,E2 -23526.08} C_VEL
LIN {X 0,Y 183.771,Z 723.808,A -85,B 0,C 180,E1 -23528.421,E2 -23528.421} C_VEL
LIN {X 0,Y 188.937,Z 713.231,A -85,B 0,C 180,E1 -23530.613,E2 -23530.613} C_VEL
LIN {X 0,Y 193.323,Z 702.825,A -85,B 0,C 180,E1 -23532.262,E2 -23532.262} C_VEL
LIN {X 0,Y 197.372,Z 691.409,A -85,B 0,C 180,E1 -23533.621,E2 -23533.621} C_VEL
LIN {X 0,Y 201.222,Z 677.784,A -85,B 0,C 180,E1 -23534.775,E2 -23534.775} C_VEL
LIN {X 0,Y 203.752,Z 665.112,A -85,B 0,C 180,E1 -23535.543,E2 -23535.543} C_VEL
LIN {X 0,Y 205.651,Z 648.314,A -85,B 0,C 180,E1 -23536.218,E2 -23536.218} C_VEL
LIN {X 0,Y 207.514,Z 627.777,A -85,B 0,C 180,E1 -23536.966,E2 -23536.966} C_VEL
LIN {X 0,Y 207.412,Z 624.742,A -85,B 0,C 180,E1 -23537.253,E2 -23537.253} C_VEL
LIN {X 0,Y 204.462,Z 615.997,A -85,B 0,C 180,E1 -23539.423,E2 -23539.423} C_VEL
LIN {X 0,Y 201.161,Z 608.071,A -85,B 0,C 180,E1 -23542.017,E2 -23542.017} C_VEL
LIN {X 0,Y 198.944,Z 603.273,A -85,B 0,C 180,E1 -23543.958,E2 -23543.958} C_VEL
LIN {X 0,Y 197.345,Z 599.908,A -85,B 0,C 180,E1 -23545.531,E2 -23545.531} C_VEL
LIN {X 0,Y 195.037,Z 595.099,A -85,B 0,C 180,E1 -23548.16,E2 -23548.16} C_VEL
LIN {X 0,Y 192.183,Z 589.471,A -85,B 0,C 180,E1 -23552.478,E2 -23552.478} C_VEL
LIN {X 0,Y 190.144,Z 585.824,A -85,B 0,C 180,E1 -23558.022,E2 -23558.022} C_VEL
LIN {X 0,Y 189.858,Z 585.064,A -85,B 0,C 180,E1 -23560.539,E2 -23560.539} C_VEL
LIN {X 0,Y 190.247,Z 585.315,A -85,B 0,C 180,E1 -23565.013,E2 -23565.013} C_VEL
LIN {X 0,Y 191.859,Z 586.263,A -85,B 0,C 180,E1 -23569.178,E2 -23569.178} C_VEL
LIN {X 0,Y 193.674,Z 589.773,A -85,B 0,C 180,E1 -23572.462,E2 -23572.462} C_VEL
LIN {X 0,Y 195.399,Z 591.551,A -85,B 0,C 180,E1 -23574.633,E2 -23574.633} C_VEL
LIN {X 0,Y 197.5,Z 594.888,A -85,B 0,C 180,E1 -23576.909,E2 -23576.909} C_VEL
LIN {X 0,Y 201.977,Z 602.305,A -85,B 0,C 180,E1 -23580.862,E2 -23580.862} C_VEL
LIN {X 0,Y 206.497,Z 610.981,A -85,B 0,C 180,E1 -23584.139,E2 -23584.139} C_VEL
LIN {X 0,Y 208.532,Z 615.235,A -85,B 0,C 180,E1 -23585.463,E2 -23585.463} C_VEL
LIN {X 0,Y 205.121,Z 649.849,A -85,B 0,C 180,E1 -23586.75,E2 -23586.75} C_VEL
LIN {X 0,Y 202.712,Z 663.927,A -85,B 0,C 180,E1 -23587.629,E2 -23587.629} C_VEL
LIN {X 0,Y 199.6,Z 676.827,A -85,B 0,C 180,E1 -23588.862,E2 -23588.862} C_VEL
LIN {X 0,Y 195.946,Z 688.38,A -85,B 0,C 180,E1 -23590.33,E2 -23590.33} C_VEL
LIN {X 0,Y 191.509,Z 699.61,A -85,B 0,C 180,E1 -23592.18,E2 -23592.18} C_VEL
LIN {X 0,Y 187.08,Z 709.089,A -85,B 0,C 180,E1 -23594.22,E2 -23594.22} C_VEL
LIN {X 0,Y 182.003,Z 718.478,A -85,B 0,C 180,E1 -23596.821,E2 -23596.821} C_VEL
LIN {X 0,Y 177.273,Z 726.129,A -85,B 0,C 180,E1 -23599.552,E2 -23599.552} C_VEL
LIN {X 0,Y 172.926,Z 732.389,A -85,B 0,C 180,E1 -23602.398,E2 -23602.398} C_VEL
LIN {X 0,Y 168.236,Z 738.48,A -85,B 0,C 180,E1 -23606.086,E2 -23606.086} C_VEL
LIN {X 0,Y 164.971,Z 742.323,A -85,B 0,C 180,E1 -23609.183,E2 -23609.183} C_VEL
LIN {X 0,Y 162.046,Z 745.388,A -85,B 0,C 180,E1 -23612.521,E2 -23612.521} C_VEL
LIN {X 0,Y 160.473,Z 746.9,A -85,B 0,C 180,E1 -23614.703,E2 -23614.703} C_VEL
LIN {X 0,Y 158.234,Z 748.679,A -85,B 0,C 180,E1 -23618.447,E2 -23618.447} C_VEL
LIN {X 0,Y 156.574,Z 749.561,A -85,B 0,C 180,E1 -23622.32,E2 -23622.32} C_VEL
LIN {X 0,Y 155.249,Z 749.401,A -85,B 0,C 180,E1 -23627.233,E2 -23627.233} C_VEL
LIN {X 0,Y 154.802,Z 748.479,A -85,B 0,C 180,E1 -23630.537,E2 -23630.537} C_VEL
LIN {X 0,Y 154.786,Z 746.344,A -85,B 0,C 180,E1 -23634.812,E2 -23634.812} C_VEL
LIN {X 0,Y 155.472,Z 742.965,A -85,B 0,C 180,E1 -23639.188,E2 -23639.188} C_VEL
LIN {X 0,Y 156.685,Z 737.91,A -85,B 0,C 180,E1 -23643.774,E2 -23643.774} C_VEL
LIN {X 0,Y 158.14,Z 732.454,A -85,B 0,C 180,E1 -23647.533,E2 -23647.533} C_VEL
LIN {X 0,Y 160.266,Z 725.158,A -85,B 0,C 180,E1 -23651.463,E2 -23651.463} C_VEL
LIN {X 0,Y 162.671,Z 716.825,A -85,B 0,C 180,E1 -23654.976,E2 -23654.976} C_VEL
LIN {X 0,Y 165.249,Z 707.714,A -85,B 0,C 180,E1 -23658.003,E2 -23658.003} C_VEL
LIN {X 0,Y 167.879,Z 697.701,A -85,B 0,C 180,E1 -23660.652,E2 -23660.652} C_VEL
LIN {X 0,Y 170.415,Z 686.983,A -85,B 0,C 180,E1 -23662.893,E2 -23662.893} C_VEL
LIN {X 0,Y 172.862,Z 674.449,A -85,B 0,C 180,E1 -23664.898,E2 -23664.898} C_VEL
LIN {X 0,Y 174.837,Z 661.831,A -85,B 0,C 180,E1 -23666.394,E2 -23666.394} C_VEL
LIN {X 0,Y 176.24,Z 648.962,A -85,B 0,C 180,E1 -23667.461,E2 -23667.461} C_VEL
LIN {X 0,Y 177.438,Z 631.356,A -85,B 0,C 180,E1 -23668.324,E2 -23668.324} C_VEL
LIN {X 0,Y 179.765,Z 594.934,A -85,B 0,C 180,E1 -23669.819,E2 -23669.819} C_VEL
LIN {X 0,Y 176.067,Z 585.615,A -85,B 0,C 180,E1 -23671.012,E2 -23671.012} C_VEL
LIN {X 0,Y 167.101,Z 566.596,A -85,B 0,C 180,E1 -23673.912,E2 -23673.912} C_VEL
LIN {X 0,Y 159.918,Z 554.298,A -85,B 0,C 180,E1 -23676.348,E2 -23676.348} C_VEL
LIN {X 0,Y 158.153,Z 551.291,A -85,B 0,C 180,E1 -23676.98,E2 -23676.98} C_VEL
LIN {X 0,Y 157.81,Z 549.827,A -85,B 0,C 180,E1 -23677.196,E2 -23677.196} C_VEL
LIN {X 0,Y 157.703,Z 549.837,A -85,B 0,C 180,E1 -23681.362,E2 -23681.362} C_VEL
LIN {X 0,Y 157.475,Z 549.866,A -85,B 0,C 180,E1 -23685.532,E2 -23685.532} C_VEL
LIN {X 0,Y 157.367,Z 549.88,A -85,B 0,C 180,E1 -23690.933,E2 -23690.933} C_VEL
LIN {X 0,Y 157.312,Z 549.886,A -85,B 0,C 180,E1 -23696.685,E2 -23696.685} C_VEL
LIN {X 0,Y 157.28,Z 549.893,A -85,B 0,C 180,E1 -23702.425,E2 -23702.425} C_VEL
LIN {X 0,Y 157.336,Z 549.885,A -85,B 0,C 180,E1 -23706.485,E2 -23706.485} C_VEL
LIN {X 0,Y 157.293,Z 549.889,A -85,B 0,C 180,E1 -23712.082,E2 -23712.082} C_VEL
LIN {X 0,Y 157.308,Z 549.883,A -85,B 0,C 180,E1 -23715.628,E2 -23715.628} C_VEL
LIN {X 0,Y 157.287,Z 549.889,A -85,B 0,C 180,E1 -23721.279,E2 -23721.279} C_VEL
LIN {X 0,Y 157.296,Z 549.889,A -85,B 0,C 180,E1 -23724.492,E2 -23724.492} C_VEL
LIN {X 0,Y 157.291,Z 549.869,A -85,B 0,C 180,E1 -23728.095,E2 -23728.095} C_VEL
LIN {X 0,Y 157.311,Z 549.89,A -85,B 0,C 180,E1 -23733.466,E2 -23733.466} C_VEL
LIN {X 0,Y 157.387,Z 549.858,A -85,B 0,C 180,E1 -23739.671,E2 -23739.671} C_VEL
LIN {X 0,Y 157.449,Z 549.87,A -85,B 0,C 180,E1 -23744.467,E2 -23744.467} C_VEL
LIN {X 0,Y 157.721,Z 549.813,A -85,B 0,C 180,E1 -23749.734,E2 -23749.734} C_VEL
LIN {X 0,Y 157.8,Z 549.815,A -85,B 0,C 180,E1 -23752.323,E2 -23752.323} C_VEL
LIN {X 0,Y 158.255,Z 549.75,A -85,B 0,C 180,E1 -23760.001,E2 -23760.001} C_VEL
LIN {X 0,Y 157.725,Z 549.836,A -85,B 0,C 180,E1 -23765.114,E2 -23765.114} C_VEL
LIN {X 0,Y 157.768,Z 549.823,A -85,B 0,C 180,E1 -23767.681,E2 -23767.681} C_VEL
LIN {X 0,Y 157.635,Z 549.84,A -85,B 0,C 180,E1 -23771.238,E2 -23771.238} C_VEL
LIN {X 0,Y 157.451,Z 549.867,A -85,B 0,C 180,E1 -23775.536,E2 -23775.536} C_VEL
LIN {X 0,Y 157.368,Z 549.883,A -85,B 0,C 180,E1 -23780.934,E2 -23780.934} C_VEL
LIN {X 0,Y 157.31,Z 549.89,A -85,B 0,C 180,E1 -23786.683,E2 -23786.683} C_VEL
LIN {X 0,Y 157.278,Z 549.895,A -85,B 0,C 180,E1 -23792.428,E2 -23792.428} C_VEL
LIN {X 0,Y 157.283,Z 549.893,A -85,B 0,C 180,E1 -23796.458,E2 -23796.458} C_VEL
LIN {X 0,Y 157.283,Z 550.017,A -85,B 0,C 180,E1 -23801.536,E2 -23801.536} C_VEL
LIN {X 0,Y 158.342,Z 554.169,A -85,B 0,C 180,E1 -23804.289,E2 -23804.289} C_VEL
LIN {X 0,Y 160.444,Z 558.475,A -85,B 0,C 180,E1 -23805.073,E2 -23805.073} C_VEL
LIN {X 0,Y 167.512,Z 574.28,A -85,B 0,C 180,E1 -23807.657,E2 -23807.657} C_VEL
LIN {X 0,Y 174.262,Z 591.841,A -85,B 0,C 180,E1 -23810.022,E2 -23810.022} C_VEL
LIN {X 0,Y 176.319,Z 598.25,A -85,B 0,C 180,E1 -23810.765,E2 -23810.765} C_VEL
LIN {X 0,Y 178.512,Z 622.639,A -85,B 0,C 180,E1 -23812.449,E2 -23812.449} C_VEL
LIN {X 0,Y 175.95,Z 664.212,A -85,B 0,C 180,E1 -23814.257,E2 -23814.257} C_VEL
LIN {X 0,Y 174.553,Z 676.744,A -85,B 0,C 180,E1 -23815.165,E2 -23815.165} C_VEL
LIN {X 0,Y 172.486,Z 689.148,A -85,B 0,C 180,E1 -23816.455,E2 -23816.455} C_VEL
LIN {X 0,Y 170.006,Z 701.214,A -85,B 0,C 180,E1 -23818.192,E2 -23818.192} C_VEL
LIN {X 0,Y 167.188,Z 712.747,A -85,B 0,C 180,E1 -23820.402,E2 -23820.402} C_VEL
LIN {X 0,Y 164.421,Z 723.207,A -85,B 0,C 180,E1 -23822.99,E2 -23822.99} C_VEL
LIN {X 0,Y 161.68,Z 732.907,A -85,B 0,C 180,E1 -23826.075,E2 -23826.075} C_VEL
LIN {X 0,Y 159.354,Z 741.023,A -85,B 0,C 180,E1 -23829.34,E2 -23829.34} C_VEL
LIN {X 0,Y 157.404,Z 748.466,A -85,B 0,C 180,E1 -23833.129,E2 -23833.129} C_VEL
LIN {X 0,Y 157.001,Z 749.868,A -85,B 0,C 180,E1 -23833.963,E2 -23833.963} C_VEL
LIN {X 0,Y 155.594,Z 752.718,A -85,B 0,C 180,E1 -23835.805,E2 -23835.805} C_VEL
LIN {X 0,Y 150.476,Z 758.042,A -85,B 0,C 180,E1 -23840.22,E2 -23840.22} C_VEL
LIN {X 0,Y 148.385,Z 760.531,A -85,B 0,C 180,E1 -23842.994,E2 -23842.994} C_VEL
LIN {X 0,Y 148.097,Z 761.646,A -85,B 0,C 180,E1 -23844.448,E2 -23844.448} C_VEL
LIN {X 0,Y 148.118,Z 763.521,A -85,B 0,C 180,E1 -23847.28,E2 -23847.28} C_VEL
LIN {X 0,Y 148.243,Z 764.827,A -85,B 0,C 180,E1 -23850,E2 -23850} C_VEL
LIN {X 0,Y 147.943,Z 765.943,A -85,B 0,C 180,E1 -23853.95,E2 -23853.95} C_VEL
LIN {X 0,Y 147.945,Z 766.188,A -85,B 0,C 180,E1 -23858.193,E2 -23858.193} C_VEL
LIN {X 0,Y 148.971,Z 765.088,A -85,B 0,C 180,E1 -23863.643,E2 -23863.643} C_VEL
LIN {X 0,Y 151.357,Z 762.491,A -85,B 0,C 180,E1 -23868.967,E2 -23868.967} C_VEL
LIN {X 0,Y 154.036,Z 759.451,A -85,B 0,C 180,E1 -23872.818,E2 -23872.818} C_VEL
LIN {X 0,Y 157.48,Z 755.427,A -85,B 0,C 180,E1 -23876.504,E2 -23876.504} C_VEL
LIN {X 0,Y 161.408,Z 750.327,A -85,B 0,C 180,E1 -23880.048,E2 -23880.048} C_VEL
LIN {X 0,Y 166.125,Z 744.03,A -85,B 0,C 180,E1 -23883.364,E2 -23883.364} C_VEL
LIN {X 0,Y 171.47,Z 736.282,A -85,B 0,C 180,E1 -23886.462,E2 -23886.462} C_VEL
LIN {X 0,Y 177.343,Z 726.677,A -85,B 0,C 180,E1 -23889.35,E2 -23889.35} C_VEL
LIN {X 0,Y 182.591,Z 716.877,A -85,B 0,C 180,E1 -23891.601,E2 -23891.601} C_VEL
LIN {X 0,Y 187.657,Z 705.996,A -85,B 0,C 180,E1 -23893.484,E2 -23893.484} C_VEL
LIN {X 0,Y 192.377,Z 693.842,A -85,B 0,C 180,E1 -23895.056,E2 -23895.056} C_VEL
LIN {X 0,Y 196.012,Z 682.539,A -85,B 0,C 180,E1 -23896.11,E2 -23896.11} C_VEL
LIN {X 0,Y 199.138,Z 669.463,A -85,B 0,C 180,E1 -23897.012,E2 -23897.012} C_VEL
LIN {X 0,Y 201.28,Z 655.238,A -85,B 0,C 180,E1 -23897.685,E2 -23897.685} C_VEL
LIN {X 0,Y 203.844,Z 628.96,A -85,B 0,C 180,E1 -23898.628,E2 -23898.628} C_VEL
LIN {X 0,Y 203.248,Z 626.348,A -85,B 0,C 180,E1 -23899.153,E2 -23899.153} C_VEL
LIN {X 0,Y 200.549,Z 618.41,A -85,B 0,C 180,E1 -23901.364,E2 -23901.364} C_VEL
LIN {X 0,Y 197.432,Z 610.735,A -85,B 0,C 180,E1 -23904.179,E2 -23904.179} C_VEL
LIN {X 0,Y 195.185,Z 605.772,A -85,B 0,C 180,E1 -23906.548,E2 -23906.548} C_VEL
LIN {X 0,Y 193.239,Z 601.464,A -85,B 0,C 180,E1 -23908.959,E2 -23908.959} C_VEL
LIN {X 0,Y 190.796,Z 596.236,A -85,B 0,C 180,E1 -23913.002,E2 -23913.002} C_VEL
LIN {X 0,Y 188.981,Z 592.564,A -85,B 0,C 180,E1 -23918.775,E2 -23918.775} C_VEL
LIN {X 0,Y 188.82,Z 592.096,A -85,B 0,C 180,E1 -23920.427,E2 -23920.427} C_VEL
LIN {X 0,Y 189.444,Z 592.498,A -85,B 0,C 180,E1 -23926.004,E2 -23926.004} C_VEL
LIN {X 0,Y 190.611,Z 593.313,A -85,B 0,C 180,E1 -23928.843,E2 -23928.843} C_VEL
LIN {X 0,Y 192.544,Z 596.903,A -85,B 0,C 180,E1 -23932.418,E2 -23932.418} C_VEL
LIN {X 0,Y 193.857,Z 598.284,A -85,B 0,C 180,E1 -23934.122,E2 -23934.122} C_VEL
LIN {X 0,Y 195.679,Z 601.46,A -85,B 0,C 180,E1 -23936.256,E2 -23936.256} C_VEL
LIN {X 0,Y 199.175,Z 607.604,A -85,B 0,C 180,E1 -23939.627,E2 -23939.627} C_VEL
LIN {X 0,Y 201.747,Z 612.615,A -85,B 0,C 180,E1 -23941.738,E2 -23941.738} C_VEL
LIN {X 0,Y 204.676,Z 618.805,A -85,B 0,C 180,E1 -23943.887,E2 -23943.887} C_VEL
LIN {X 0,Y 201.412,Z 650.341,A -85,B 0,C 180,E1 -23945.057,E2 -23945.057} C_VEL
LIN {X 0,Y 198.939,Z 664.164,A -85,B 0,C 180,E1 -23945.91,E2 -23945.91} C_VEL
LIN {X 0,Y 196.041,Z 675.861,A -85,B 0,C 180,E1 -23947,E2 -23947} C_VEL
LIN {X 0,Y 192.34,Z 687.266,A -85,B 0,C 180,E1 -23948.403,E2 -23948.403} C_VEL
LIN {X 0,Y 187.506,Z 699.173,A -85,B 0,C 180,E1 -23950.312,E2 -23950.312} C_VEL
LIN {X 0,Y 182.637,Z 709.261,A -85,B 0,C 180,E1 -23952.466,E2 -23952.466} C_VEL
LIN {X 0,Y 177.352,Z 718.53,A -85,B 0,C 180,E1 -23955.007,E2 -23955.007} C_VEL
LIN {X 0,Y 171.858,Z 726.976,A -85,B 0,C 180,E1 -23958.054,E2 -23958.054} C_VEL
LIN {X 0,Y 166.306,Z 734.314,A -85,B 0,C 180,E1 -23961.614,E2 -23961.614} C_VEL
LIN {X 0,Y 162.374,Z 739.017,A -85,B 0,C 180,E1 -23964.644,E2 -23964.644} C_VEL
LIN {X 0,Y 158.909,Z 742.818,A -85,B 0,C 180,E1 -23967.808,E2 -23967.808} C_VEL
LIN {X 0,Y 155.906,Z 745.734,A -85,B 0,C 180,E1 -23971.077,E2 -23971.077} C_VEL
LIN {X 0,Y 153.389,Z 747.865,A -85,B 0,C 180,E1 -23974.441,E2 -23974.441} C_VEL
LIN {X 0,Y 151.335,Z 749.291,A -85,B 0,C 180,E1 -23977.865,E2 -23977.865} C_VEL
LIN {X 0,Y 149.79,Z 749.993,A -85,B 0,C 180,E1 -23981.35,E2 -23981.35} C_VEL
LIN {X 0,Y 148.576,Z 749.997,A -85,B 0,C 180,E1 -23985.195,E2 -23985.195} C_VEL
LIN {X 0,Y 147.78,Z 749.062,A -85,B 0,C 180,E1 -23989.542,E2 -23989.542} C_VEL
LIN {X 0,Y 147.655,Z 747.039,A -85,B 0,C 180,E1 -23994.011,E2 -23994.011} C_VEL
LIN {X 0,Y 148.218,Z 743.787,A -85,B 0,C 180,E1 -23998.592,E2 -23998.592} C_VEL
LIN {X 0,Y 149.402,Z 738.987,A -85,B 0,C 180,E1 -24003.348,E2 -24003.348} C_VEL
LIN {X 0,Y 150.904,Z 733.504,A -85,B 0,C 180,E1 -24007.405,E2 -24007.405} C_VEL
LIN {X 0,Y 153.201,Z 725.834,A -85,B 0,C 180,E1 -24011.78,E2 -24011.78} C_VEL
LIN {X 0,Y 155.278,Z 718.885,A -85,B 0,C 180,E1 -24014.916,E2 -24014.916} C_VEL
LIN {X 0,Y 157.973,Z 709.953,A -85,B 0,C 180,E1 -24018.159,E2 -24018.159} C_VEL
LIN {X 0,Y 160.921,Z 699.203,A -85,B 0,C 180,E1 -24021.208,E2 -24021.208} C_VEL
LIN {X 0,Y 163.911,Z 687.142,A -85,B 0,C 180,E1 -24023.847,E2 -24023.847} C_VEL
LIN {X 0,Y 166.43,Z 674.581,A -85,B 0,C 180,E1 -24025.914,E2 -24025.914} C_VEL
LIN {X 0,Y 168.522,Z 661.814,A -85,B 0,C 180,E1 -24027.46,E2 -24027.46} C_VEL
LIN {X 0,Y 169.894,Z 649.474,A -85,B 0,C 180,E1 -24028.513,E2 -24028.513} C_VEL
LIN {X 0,Y 171.187,Z 631.644,A -85,B 0,C 180,E1 -24029.413,E2 -24029.413} C_VEL
LIN {X 0,Y 173.481,Z 596.623,A -85,B 0,C 180,E1 -24030.9,E2 -24030.9} C_VEL
LIN {X 0,Y 170.232,Z 588.541,A -85,B 0,C 180,E1 -24031.984,E2 -24031.984} C_VEL
LIN {X 0,Y 161.856,Z 570.519,A -85,B 0,C 180,E1 -24034.877,E2 -24034.877} C_VEL
LIN {X 0,Y 152.329,Z 554.341,A -85,B 0,C 180,E1 -24038.323,E2 -24038.323} C_VEL
LIN {X 0,Y 150.969,Z 551.903,A -85,B 0,C 180,E1 -24038.871,E2 -24038.871} C_VEL
LIN {X 0,Y 150.718,Z 550.709,A -85,B 0,C 180,E1 -24039.054,E2 -24039.054} C_VEL
LIN {X 0,Y 150.461,Z 550.739,A -85,B 0,C 180,E1 -24043.506,E2 -24043.506} C_VEL
LIN {X 0,Y 150.364,Z 550.751,A -85,B 0,C 180,E1 -24049.097,E2 -24049.097} C_VEL
LIN {X 0,Y 150.223,Z 550.771,A -85,B 0,C 180,E1 -24054.9,E2 -24054.9} C_VEL
LIN {X 0,Y 150.219,Z 550.772,A -85,B 0,C 180,E1 -24057.894,E2 -24057.894} C_VEL
LIN {X 0,Y 150.222,Z 550.771,A -85,B 0,C 180,E1 -24062.639,E2 -24062.639} C_VEL
LIN {X 0,Y 150.266,Z 550.759,A -85,B 0,C 180,E1 -24067.445,E2 -24067.445} C_VEL
LIN {X 0,Y 150.234,Z 550.767,A -85,B 0,C 180,E1 -24071.543,E2 -24071.543} C_VEL
LIN {X 0,Y 150.258,Z 550.762,A -85,B 0,C 180,E1 -24075.447,E2 -24075.447} C_VEL
LIN {X 0,Y 150.231,Z 550.754,A -85,B 0,C 180,E1 -24079.087,E2 -24079.087} C_VEL
LIN {X 0,Y 150.238,Z 550.769,A -85,B 0,C 180,E1 -24082.677,E2 -24082.677} C_VEL
LIN {X 0,Y 150.216,Z 550.751,A -85,B 0,C 180,E1 -24087.365,E2 -24087.365} C_VEL
LIN {X 0,Y 150.237,Z 550.769,A -85,B 0,C 180,E1 -24092.721,E2 -24092.721} C_VEL
LIN {X 0,Y 150.345,Z 550.734,A -85,B 0,C 180,E1 -24099.211,E2 -24099.211} C_VEL
LIN {X 0,Y 150.357,Z 550.753,A -85,B 0,C 180,E1 -24103.714,E2 -24103.714} C_VEL
LIN {X 0,Y 150.647,Z 550.696,A -85,B 0,C 180,E1 -24109.246,E2 -24109.246} C_VEL
LIN {X 0,Y 150.735,Z 550.69,A -85,B 0,C 180,E1 -24111.961,E2 -24111.961} C_VEL
LIN {X 0,Y 151.216,Z 550.626,A -85,B 0,C 180,E1 -24120.001,E2 -24120.001} C_VEL
LIN {X 0,Y 150.67,Z 550.714,A -85,B 0,C 180,E1 -24125.354,E2 -24125.354} C_VEL
LIN {X 0,Y 150.705,Z 550.701,A -85,B 0,C 180,E1 -24128.044,E2 -24128.044} C_VEL
LIN {X 0,Y 150.575,Z 550.72,A -85,B 0,C 180,E1 -24131.439,E2 -24131.439} C_VEL
LIN {X 0,Y 150.358,Z 550.748,A -85,B 0,C 180,E1 -24136.288,E2 -24136.288} C_VEL
LIN {X 0,Y 150.349,Z 550.757,A -85,B 0,C 180,E1 -24140.793,E2 -24140.793} C_VEL
LIN {X 0,Y 150.241,Z 550.772,A -85,B 0,C 180,E1 -24147.282,E2 -24147.282} C_VEL
LIN {X 0,Y 150.218,Z 550.774,A -85,B 0,C 180,E1 -24152.636,E2 -24152.636} C_VEL
LIN {X 0,Y 150.212,Z 550.771,A -85,B 0,C 180,E1 -24157.464,E2 -24157.464} C_VEL
LIN {X 0,Y 150.217,Z 550.827,A -85,B 0,C 180,E1 -24160.259,E2 -24160.259} C_VEL
LIN {X 0,Y 150.963,Z 553.748,A -85,B 0,C 180,E1 -24162.299,E2 -24162.299} C_VEL
LIN {X 0,Y 158.043,Z 568.481,A -85,B 0,C 180,E1 -24165.116,E2 -24165.116} C_VEL
LIN {X 0,Y 164.342,Z 583.607,A -85,B 0,C 180,E1 -24167.516,E2 -24167.516} C_VEL
LIN {X 0,Y 170.233,Z 599.944,A -85,B 0,C 180,E1 -24169.684,E2 -24169.684} C_VEL
LIN {X 0,Y 172.261,Z 623.287,A -85,B 0,C 180,E1 -24171.363,E2 -24171.363} C_VEL
LIN {X 0,Y 169.667,Z 663.832,A -85,B 0,C 180,E1 -24173.179,E2 -24173.179} C_VEL
LIN {X 0,Y 168.203,Z 676.338,A -85,B 0,C 180,E1 -24174.109,E2 -24174.109} C_VEL
LIN {X 0,Y 165.98,Z 689.301,A -85,B 0,C 180,E1 -24175.506,E2 -24175.506} C_VEL
LIN {X 0,Y 163.594,Z 700.406,A -85,B 0,C 180,E1 -24177.156,E2 -24177.156} C_VEL
LIN {X 0,Y 161.038,Z 710.715,A -85,B 0,C 180,E1 -24179.151,E2 -24179.151} C_VEL
LIN {X 0,Y 158.092,Z 721.433,A -85,B 0,C 180,E1 -24181.815,E2 -24181.815} C_VEL
LIN {X 0,Y 155.443,Z 730.63,A -85,B 0,C 180,E1 -24184.726,E2 -24184.726} C_VEL
LIN {X 0,Y 153.093,Z 738.291,A -85,B 0,C 180,E1 -24187.746,E2 -24187.746} C_VEL
LIN {X 0,Y 150.914,Z 746.193,A -85,B 0,C 180,E1 -24191.679,E2 -24191.679} C_VEL
LIN {X 0,Y 149.035,Z 753.378,A -85,B 0,C 180,E1 -24196.363,E2 -24196.363} C_VEL
LIN {X 0,Y 148.266,Z 758.14,A -85,B 0,C 180,E1 -24200.45,E2 -24200.45} C_VEL
LIN {X 0,Y 148.097,Z 761.646,A -85,B 0,C 180,E1 -24204.448,E2 -24204.448} C_VEL
LIN {X 0,Y 147.807,Z 762.689,A -85,B 0,C 180,E1 -24205.911,E2 -24205.911} C_VEL
LIN {X 0,Y 146.98,Z 763.541,A -85,B 0,C 180,E1 -24207.372,E2 -24207.372} C_VEL
LIN {X 0,Y 144.47,Z 764.735,A -85,B 0,C 180,E1 -24210.307,E2 -24210.307} C_VEL
LIN {X 0,Y 141.915,Z 765.39,A -85,B 0,C 180,E1 -24213.381,E2 -24213.381} C_VEL
LIN {X 0,Y 140.845,Z 765.644,A -85,B 0,C 180,E1 -24215.794,E2 -24215.794} C_VEL
LIN {X 0,Y 140.773,Z 765.668,A -85,B 0,C 180,E1 -24216.615,E2 -24216.615} C_VEL
LIN {X 0,Y 141.316,Z 765.491,A -85,B 0,C 180,E1 -24221.474,E2 -24221.474} C_VEL
LIN {X 0,Y 143.106,Z 763.768,A -85,B 0,C 180,E1 -24227.137,E2 -24227.137} C_VEL
LIN {X 0,Y 146.459,Z 760.524,A -85,B 0,C 180,E1 -24232.574,E2 -24232.574} C_VEL
LIN {X 0,Y 149.89,Z 756.968,A -85,B 0,C 180,E1 -24236.45,E2 -24236.45} C_VEL
LIN {X 0,Y 153.821,Z 752.407,A -85,B 0,C 180,E1 -24240.17,E2 -24240.17} C_VEL
LIN {X 0,Y 159.39,Z 745.633,A -85,B 0,C 180,E1 -24244.206,E2 -24244.206} C_VEL
LIN {X 0,Y 164.912,Z 738.324,A -85,B 0,C 180,E1 -24247.392,E2 -24247.392} C_VEL
LIN {X 0,Y 169.86,Z 730.98,A -85,B 0,C 180,E1 -24249.889,E2 -24249.889} C_VEL
LIN {X 0,Y 175.157,Z 722.225,A -85,B 0,C 180,E1 -24252.226,E2 -24252.226} C_VEL
LIN {X 0,Y 180.905,Z 711.544,A -85,B 0,C 180,E1 -24254.368,E2 -24254.368} C_VEL
LIN {X 0,Y 185.669,Z 700.992,A -85,B 0,C 180,E1 -24255.986,E2 -24255.986} C_VEL
LIN {X 0,Y 190.075,Z 689.341,A -85,B 0,C 180,E1 -24257.295,E2 -24257.295} C_VEL
LIN {X 0,Y 193.803,Z 676.834,A -85,B 0,C 180,E1 -24258.326,E2 -24258.326} C_VEL
LIN {X 0,Y 196.598,Z 663.875,A -85,B 0,C 180,E1 -24259.074,E2 -24259.074} C_VEL
LIN {X 0,Y 198.502,Z 648.556,A -85,B 0,C 180,E1 -24259.69,E2 -24259.69} C_VEL
LIN {X 0,Y 200.213,Z 631.277,A -85,B 0,C 180,E1 -24260.325,E2 -24260.325} C_VEL
LIN {X 0,Y 198.025,Z 624.192,A -85,B 0,C 180,E1 -24262.34,E2 -24262.34} C_VEL
LIN {X 0,Y 195.312,Z 616.842,A -85,B 0,C 180,E1 -24265.029,E2 -24265.029} C_VEL
LIN {X 0,Y 193.218,Z 611.929,A -85,B 0,C 180,E1 -24267.429,E2 -24267.429} C_VEL
LIN {X 0,Y 191.545,Z 607.858,A -85,B 0,C 180,E1 -24269.745,E2 -24269.745} C_VEL
LIN {X 0,Y 189.454,Z 602.946,A -85,B 0,C 180,E1 -24273.566,E2 -24273.566} C_VEL
LIN {X 0,Y 187.877,Z 599.41,A -85,B 0,C 180,E1 -24279.255,E2 -24279.255} C_VEL
LIN {X 0,Y 187.88,Z 599.145,A -85,B 0,C 180,E1 -24283.477,E2 -24283.477} C_VEL
LIN {X 0,Y 189.345,Z 600.221,A -85,B 0,C 180,E1 -24288.417,E2 -24288.417} C_VEL
LIN {X 0,Y 191.309,Z 603.886,A -85,B 0,C 180,E1 -24292.219,E2 -24292.219} C_VEL
LIN {X 0,Y 192.411,Z 605.159,A -85,B 0,C 180,E1 -24293.708,E2 -24293.708} C_VEL
LIN {X 0,Y 194.062,Z 608.328,A -85,B 0,C 180,E1 -24295.789,E2 -24295.789} C_VEL
LIN {X 0,Y 197.559,Z 614.773,A -85,B 0,C 180,E1 -24299.322,E2 -24299.322} C_VEL
LIN {X 0,Y 200.95,Z 622.017,A -85,B 0,C 180,E1 -24302.176,E2 -24302.176} C_VEL
LIN {X 0,Y 197.854,Z 650.98,A -85,B 0,C 180,E1 -24303.304,E2 -24303.304} C_VEL
LIN {X 0,Y 195.372,Z 664.37,A -85,B 0,C 180,E1 -24304.125,E2 -24304.125} C_VEL
LIN {X 0,Y 192.436,Z 675.906,A -85,B 0,C 180,E1 -24305.184,E2 -24305.184} C_VEL
LIN {X 0,Y 188.253,Z 688.21,A -85,B 0,C 180,E1 -24306.681,E2 -24306.681} C_VEL
LIN {X 0,Y 183.208,Z 700.041,A -85,B 0,C 180,E1 -24308.586,E2 -24308.586} C_VEL
LIN {X 0,Y 177.961,Z 710.247,A -85,B 0,C 180,E1 -24310.798,E2 -24310.798} C_VEL
LIN {X 0,Y 172.34,Z 719.517,A -85,B 0,C 180,E1 -24313.395,E2 -24313.395} C_VEL
LIN {X 0,Y 167.091,Z 727.12,A -85,B 0,C 180,E1 -24316.177,E2 -24316.177} C_VEL
LIN {X 0,Y 161.355,Z 734.35,A -85,B 0,C 180,E1 -24319.672,E2 -24319.672} C_VEL
LIN {X 0,Y 156.927,Z 739.31,A -85,B 0,C 180,E1 -24322.866,E2 -24322.866} C_VEL
LIN {X 0,Y 153.006,Z 743.283,A -85,B 0,C 180,E1 -24326.257,E2 -24326.257} C_VEL
LIN {X 0,Y 149.679,Z 746.244,A -85,B 0,C 180,E1 -24329.704,E2 -24329.704} C_VEL
LIN {X 0,Y 145.493,Z 749.302,A -85,B 0,C 180,E1 -24335.425,E2 -24335.425} C_VEL
LIN {X 0,Y 143.317,Z 750.341,A -85,B 0,C 180,E1 -24339.603,E2 -24339.603} C_VEL
LIN {X 0,Y 141.802,Z 750.469,A -85,B 0,C 180,E1 -24343.935,E2 -24343.935} C_VEL
LIN {X 0,Y 140.707,Z 749.297,A -85,B 0,C 180,E1 -24349.511,E2 -24349.511} C_VEL
LIN {X 0,Y 140.614,Z 746.712,A -85,B 0,C 180,E1 -24354.93,E2 -24354.93} C_VEL
LIN {X 0,Y 141.468,Z 742.667,A -85,B 0,C 180,E1 -24360.213,E2 -24360.213} C_VEL
LIN {X 0,Y 142.892,Z 737.195,A -85,B 0,C 180,E1 -24365.288,E2 -24365.288} C_VEL
LIN {X 0,Y 144.995,Z 730.026,A -85,B 0,C 180,E1 -24370.167,E2 -24370.167} C_VEL
LIN {X 0,Y 147.415,Z 722.552,A -85,B 0,C 180,E1 -24374.09,E2 -24374.09} C_VEL
LIN {X 0,Y 149.935,Z 714.487,A -85,B 0,C 180,E1 -24377.46,E2 -24377.46} C_VEL
LIN {X 0,Y 152.872,Z 704.521,A -85,B 0,C 180,E1 -24380.741,E2 -24380.741} C_VEL
LIN {X 0,Y 155.883,Z 693.543,A -85,B 0,C 180,E1 -24383.553,E2 -24383.553} C_VEL
LIN {X 0,Y 158.647,Z 681.804,A -85,B 0,C 180,E1 -24385.872,E2 -24385.872} C_VEL
LIN {X 0,Y 161.046,Z 669.266,A -85,B 0,C 180,E1 -24387.73,E2 -24387.73} C_VEL
LIN {X 0,Y 162.934,Z 656.006,A -85,B 0,C 180,E1 -24389.155,E2 -24389.155} C_VEL
LIN {X 0,Y 164.277,Z 642.014,A -85,B 0,C 180,E1 -24390.104,E2 -24390.104} C_VEL
LIN {X 0,Y 167.294,Z 598.247,A -85,B 0,C 180,E1 -24392.029,E2 -24392.029} C_VEL
LIN {X 0,Y 163.126,Z 588.664,A -85,B 0,C 180,E1 -24393.485,E2 -24393.485} C_VEL
LIN {X 0,Y 156.763,Z 574.669,A -85,B 0,C 180,E1 -24395.835,E2 -24395.835} C_VEL
LIN {X 0,Y 147.471,Z 558.818,A -85,B 0,C 180,E1 -24399.4,E2 -24399.4} C_VEL
LIN {X 0,Y 145.678,Z 555.738,A -85,B 0,C 180,E1 -24400.154,E2 -24400.154} C_VEL
LIN {X 0,Y 143.991,Z 553.112,A -85,B 0,C 180,E1 -24400.862,E2 -24400.862} C_VEL
LIN {X 0,Y 143.637,Z 551.59,A -85,B 0,C 180,E1 -24401.108,E2 -24401.108} C_VEL
LIN {X 0,Y 143.314,Z 551.628,A -85,B 0,C 180,E1 -24407.111,E2 -24407.111} C_VEL
LIN {X 0,Y 143.274,Z 551.636,A -85,B 0,C 180,E1 -24411.255,E2 -24411.255} C_VEL
LIN {X 0,Y 143.187,Z 551.648,A -85,B 0,C 180,E1 -24417.937,E2 -24417.937} C_VEL
LIN {X 0,Y 143.175,Z 551.648,A -85,B 0,C 180,E1 -24423.441,E2 -24423.441} C_VEL
LIN {X 0,Y 143.138,Z 551.641,A -85,B 0,C 180,E1 -24429.664,E2 -24429.664} C_VEL
LIN {X 0,Y 143.179,Z 551.65,A -85,B 0,C 180,E1 -24433.407,E2 -24433.407} C_VEL
LIN {X 0,Y 143.159,Z 551.632,A -85,B 0,C 180,E1 -24437.423,E2 -24437.423} C_VEL
LIN {X 0,Y 143.165,Z 551.65,A -85,B 0,C 180,E1 -24441.76,E2 -24441.76} C_VEL
LIN {X 0,Y 143.184,Z 551.627,A -85,B 0,C 180,E1 -24447.323,E2 -24447.323} C_VEL
LIN {X 0,Y 143.184,Z 551.647,A -85,B 0,C 180,E1 -24452.065,E2 -24452.065} C_VEL
LIN {X 0,Y 143.271,Z 551.615,A -85,B 0,C 180,E1 -24458.749,E2 -24458.749} C_VEL
LIN {X 0,Y 143.297,Z 551.629,A -85,B 0,C 180,E1 -24462.888,E2 -24462.888} C_VEL
LIN {X 0,Y 143.591,Z 551.578,A -85,B 0,C 180,E1 -24468.711,E2 -24468.711} C_VEL
LIN {X 0,Y 143.656,Z 551.567,A -85,B 0,C 180,E1 -24471.562,E2 -24471.562} C_VEL
LIN {X 0,Y 144.175,Z 551.502,A -85,B 0,C 180,E1 -24480.001,E2 -24480.001} C_VEL
LIN {X 0,Y 143.614,Z 551.592,A -85,B 0,C 180,E1 -24485.618,E2 -24485.618} C_VEL
LIN {X 0,Y 143.626,Z 551.58,A -85,B 0,C 180,E1 -24488.443,E2 -24488.443} C_VEL
LIN {X 0,Y 143.503,Z 551.602,A -85,B 0,C 180,E1 -24491.631,E2 -24491.631} C_VEL
LIN {X 0,Y 143.298,Z 551.623,A -85,B 0,C 180,E1 -24497.115,E2 -24497.115} C_VEL
LIN {X 0,Y 143.275,Z 551.639,A -85,B 0,C 180,E1 -24501.255,E2 -24501.255} C_VEL
LIN {X 0,Y 143.188,Z 551.648,A -85,B 0,C 180,E1 -24507.937,E2 -24507.937} C_VEL
LIN {X 0,Y 143.169,Z 551.647,A -85,B 0,C 180,E1 -24513.437,E2 -24513.437} C_VEL
LIN {X 0,Y 143.162,Z 551.729,A -85,B 0,C 180,E1 -24518.924,E2 -24518.924} C_VEL
LIN {X 0,Y 143.634,Z 553.464,A -85,B 0,C 180,E1 -24520.073,E2 -24520.073} C_VEL
LIN {X 0,Y 145.798,Z 557.689,A -85,B 0,C 180,E1 -24521.056,E2 -24521.056} C_VEL
LIN {X 0,Y 152.27,Z 571.035,A -85,B 0,C 180,E1 -24523.816,E2 -24523.816} C_VEL
LIN {X 0,Y 158.51,Z 586.06,A -85,B 0,C 180,E1 -24526.326,E2 -24526.326} C_VEL
LIN {X 0,Y 164.146,Z 601.75,A -85,B 0,C 180,E1 -24528.549,E2 -24528.549} C_VEL
LIN {X 0,Y 166.029,Z 624.144,A -85,B 0,C 180,E1 -24530.231,E2 -24530.231} C_VEL
LIN {X 0,Y 163.304,Z 664.201,A -85,B 0,C 180,E1 -24532.096,E2 -24532.096} C_VEL
LIN {X 0,Y 161.718,Z 677.054,A -85,B 0,C 180,E1 -24533.112,E2 -24533.112} C_VEL
LIN {X 0,Y 159.308,Z 690.179,A -85,B 0,C 180,E1 -24534.619,E2 -24534.619} C_VEL
LIN {X 0,Y 156.506,Z 702.567,A -85,B 0,C 180,E1 -24536.627,E2 -24536.627} C_VEL
LIN {X 0,Y 153.508,Z 713.699,A -85,B 0,C 180,E1 -24539,E2 -24539} C_VEL
LIN {X 0,Y 150.893,Z 722.776,A -85,B 0,C 180,E1 -24541.485,E2 -24541.485} C_VEL
LIN {X 0,Y 148.011,Z 732.081,A -85,B 0,C 180,E1 -24544.701,E2 -24544.701} C_VEL
LIN {X 0,Y 145.234,Z 741.134,A -85,B 0,C 180,E1 -24548.72,E2 -24548.72} C_VEL
LIN {X 0,Y 143.138,Z 748.386,A -85,B 0,C 180,E1 -24552.867,E2 -24552.867} C_VEL
LIN {X 0,Y 141.741,Z 754.123,A -85,B 0,C 180,E1 -24557.108,E2 -24557.108} C_VEL
LIN {X 0,Y 141.093,Z 758.607,A -85,B 0,C 180,E1 -24561.406,E2 -24561.406} C_VEL
LIN {X 0,Y 141.042,Z 761.678,A -85,B 0,C 180,E1 -24565.276,E2 -24565.276} C_VEL
LIN {X 0,Y 141.178,Z 764.223,A -85,B 0,C 180,E1 -24570,E2 -24570} C_VEL
LIN {X 0,Y 140.872,Z 765.346,A -85,B 0,C 180,E1 -24573.794,E2 -24573.794} C_VEL
LIN {X 0,Y 140.773,Z 765.668,A -85,B 0,C 180,E1 -24576.615,E2 -24576.615} C_VEL
LIN {X 0,Y 140.246,Z 765.709,A -85,B 0,C 180,E1 -24579.016,E2 -24579.016} C_VEL
LIN {X 0,Y 138.057,Z 765.078,A -85,B 0,C 180,E1 -24582.999,E2 -24582.999} C_VEL
LIN {X 0,Y 136.554,Z 763.915,A -85,B 0,C 180,E1 -24587.066,E2 -24587.066} C_VEL
LIN {X 0,Y 137.104,Z 762.867,A -85,B 0,C 180,E1 -24589.495,E2 -24589.495} C_VEL
LIN {X 0,Y 141.027,Z 759.436,A -85,B 0,C 180,E1 -24595.061,E2 -24595.061} C_VEL
LIN {X 0,Y 145.403,Z 755.127,A -85,B 0,C 180,E1 -24599.536,E2 -24599.536} C_VEL
LIN {X 0,Y 150.947,Z 749.097,A -85,B 0,C 180,E1 -24603.966,E2 -24603.966} C_VEL
LIN {X 0,Y 157.33,Z 741.529,A -85,B 0,C 180,E1 -24607.894,E2 -24607.894} C_VEL
LIN {X 0,Y 163.455,Z 733.442,A -85,B 0,C 180,E1 -24610.971,E2 -24610.971} C_VEL
LIN {X 0,Y 170.043,Z 723.484,A -85,B 0,C 180,E1 -24613.81,E2 -24613.81} C_VEL
LIN {X 0,Y 175.943,Z 713.143,A -85,B 0,C 180,E1 -24615.971,E2 -24615.971} C_VEL
LIN {X 0,Y 181.53,Z 701.64,A -85,B 0,C 180,E1 -24617.767,E2 -24617.767} C_VEL
LIN {X 0,Y 186.06,Z 690.382,A -85,B 0,C 180,E1 -24619.064,E2 -24619.064} C_VEL
LIN {X 0,Y 190.406,Z 676.62,A -85,B 0,C 180,E1 -24620.191,E2 -24620.191} C_VEL
LIN {X 0,Y 193.287,Z 663.939,A -85,B 0,C 180,E1 -24620.922,E2 -24620.922} C_VEL
LIN {X 0,Y 195.341,Z 648.495,A -85,B 0,C 180,E1 -24621.539,E2 -24621.539} C_VEL
LIN {X 0,Y 196.824,Z 634.202,A -85,B 0,C 180,E1 -24622.068,E2 -24622.068} C_VEL
LIN {X 0,Y 194.418,Z 626.421,A -85,B 0,C 180,E1 -24624.544,E2 -24624.544} C_VEL
LIN {X 0,Y 192.11,Z 620.014,A -85,B 0,C 180,E1 -24627.288,E2 -24627.288} C_VEL
LIN {X 0,Y 189.83,Z 614.106,A -85,B 0,C 180,E1 -24630.642,E2 -24630.642} C_VEL
LIN {X 0,Y 188.148,Z 609.731,A -85,B 0,C 180,E1 -24634.085,E2 -24634.085} C_VEL
LIN {X 0,Y 186.785,Z 606.328,A -85,B 0,C 180,E1 -24639.667,E2 -24639.667} C_VEL
LIN {X 0,Y 186.823,Z 606.135,A -85,B 0,C 180,E1 -24643.381,E2 -24643.381} C_VEL
LIN {X 0,Y 188.083,Z 607.076,A -85,B 0,C 180,E1 -24647.955,E2 -24647.955} C_VEL
LIN {X 0,Y 189.887,Z 610.66,A -85,B 0,C 180,E1 -24651.739,E2 -24651.739} C_VEL
LIN {X 0,Y 190.889,Z 611.872,A -85,B 0,C 180,E1 -24653.167,E2 -24653.167} C_VEL
LIN {X 0,Y 192.155,Z 614.57,A -85,B 0,C 180,E1 -24654.949,E2 -24654.949} C_VEL
LIN {X 0,Y 195.309,Z 620.71,A -85,B 0,C 180,E1 -24658.396,E2 -24658.396} C_VEL
LIN {X 0,Y 197.553,Z 625.802,A -85,B 0,C 180,E1 -24660.487,E2 -24660.487} C_VEL
LIN {X 0,Y 194.727,Z 650.961,A -85,B 0,C 180,E1 -24661.443,E2 -24661.443} C_VEL
LIN {X 0,Y 192.076,Z 664.666,A -85,B 0,C 180,E1 -24662.259,E2 -24662.259} C_VEL
LIN {X 0,Y 188.778,Z 676.907,A -85,B 0,C 180,E1 -24663.381,E2 -24663.381} C_VEL
LIN {X 0,Y 184.31,Z 689.309,A -85,B 0,C 180,E1 -24664.899,E2 -24664.899} C_VEL
LIN {X 0,Y 179.155,Z 700.768,A -85,B 0,C 180,E1 -24666.757,E2 -24666.757} C_VEL
LIN {X 0,Y 173.353,Z 711.464,A -85,B 0,C 180,E1 -24669.093,E2 -24669.093} C_VEL
LIN {X 0,Y 167.237,Z 720.95,A -85,B 0,C 180,E1 -24671.801,E2 -24671.801} C_VEL
LIN {X 0,Y 161.634,Z 728.463,A -85,B 0,C 180,E1 -24674.669,E2 -24674.669} C_VEL
LIN {X 0,Y 155.465,Z 735.627,A -85,B 0,C 180,E1 -24678.321,E2 -24678.321} C_VEL
LIN {X 0,Y 150.342,Z 740.866,A -85,B 0,C 180,E1 -24681.959,E2 -24681.959} C_VEL
LIN {X 0,Y 146.055,Z 744.75,A -85,B 0,C 180,E1 -24685.661,E2 -24685.661} C_VEL
LIN {X 0,Y 142.369,Z 747.647,A -85,B 0,C 180,E1 -24689.579,E2 -24689.579} C_VEL
LIN {X 0,Y 139.3,Z 749.631,A -85,B 0,C 180,E1 -24693.707,E2 -24693.707} C_VEL
LIN {X 0,Y 136.253,Z 750.891,A -85,B 0,C 180,E1 -24699.313,E2 -24699.313} C_VEL
LIN {X 0,Y 134.889,Z 750.886,A -85,B 0,C 180,E1 -24703.163,E2 -24703.163} C_VEL
LIN {X 0,Y 133.919,Z 750.193,A -85,B 0,C 180,E1 -24707.281,E2 -24707.281} C_VEL
LIN {X 0,Y 133.422,Z 748.375,A -85,B 0,C 180,E1 -24712.194,E2 -24712.194} C_VEL
LIN {X 0,Y 133.76,Z 745.381,A -85,B 0,C 180,E1 -24717.208,E2 -24717.208} C_VEL
LIN {X 0,Y 134.857,Z 740.963,A -85,B 0,C 180,E1 -24722.365,E2 -24722.365} C_VEL
LIN {X 0,Y 136.283,Z 735.936,A -85,B 0,C 180,E1 -24726.766,E2 -24726.766} C_VEL
LIN {X 0,Y 138.476,Z 728.932,A -85,B 0,C 180,E1 -24731.507,E2 -24731.507} C_VEL
LIN {X 0,Y 141.051,Z 721.113,A -85,B 0,C 180,E1 -24735.574,E2 -24735.574} C_VEL
LIN {X 0,Y 144.217,Z 711.508,A -85,B 0,C 180,E1 -24739.471,E2 -24739.471} C_VEL
LIN {X 0,Y 147.197,Z 701.704,A -85,B 0,C 180,E1 -24742.579,E2 -24742.579} C_VEL
LIN {X 0,Y 150.192,Z 690.633,A -85,B 0,C 180,E1 -24745.303,E2 -24745.303} C_VEL
LIN {X 0,Y 152.983,Z 678.645,A -85,B 0,C 180,E1 -24747.573,E2 -24747.573} C_VEL
LIN {X 0,Y 155.388,Z 665.609,A -85,B 0,C 180,E1 -24749.387,E2 -24749.387} C_VEL
LIN {X 0,Y 157.224,Z 651.677,A -85,B 0,C 180,E1 -24750.746,E2 -24750.746} C_VEL
LIN {X 0,Y 158.472,Z 636.946,A -85,B 0,C 180,E1 -24751.592,E2 -24751.592} C_VEL
LIN {X 0,Y 161.027,Z 599.765,A -85,B 0,C 180,E1 -24753.285,E2 -24753.285} C_VEL
LIN {X 0,Y 151.687,Z 578.828,A -85,B 0,C 180,E1 -24756.852,E2 -24756.852} C_VEL
LIN {X 0,Y 141.277,Z 560.745,A -85,B 0,C 180,E1 -24761.151,E2 -24761.151} C_VEL
LIN {X 0,Y 139.145,Z 557.28,A -85,B 0,C 180,E1 -24762.11,E2 -24762.11} C_VEL
LIN {X 0,Y 137.055,Z 554.707,A -85,B 0,C 180,E1 -24763.027,E2 -24763.027} C_VEL
LIN {X 0,Y 136.381,Z 552.492,A -85,B 0,C 180,E1 -24763.56,E2 -24763.56} C_VEL
LIN {X 0,Y 136.249,Z 552.51,A -85,B 0,C 180,E1 -24768.028,E2 -24768.028} C_VEL
LIN {X 0,Y 136.195,Z 552.516,A -85,B 0,C 180,E1 -24771.749,E2 -24771.749} C_VEL
LIN {X 0,Y 136.113,Z 552.529,A -85,B 0,C 180,E1 -24778.629,E2 -24778.629} C_VEL
LIN {X 0,Y 136.089,Z 552.533,A -85,B 0,C 180,E1 -24784.615,E2 -24784.615} C_VEL
LIN {X 0,Y 136.114,Z 552.514,A -85,B 0,C 180,E1 -24789.243,E2 -24789.243} C_VEL
LIN {X 0,Y 136.112,Z 552.529,A -85,B 0,C 180,E1 -24793.71,E2 -24793.71} C_VEL
LIN {X 0,Y 136.107,Z 552.509,A -85,B 0,C 180,E1 -24797.837,E2 -24797.837} C_VEL
LIN {X 0,Y 136.116,Z 552.528,A -85,B 0,C 180,E1 -24801.716,E2 -24801.716} C_VEL
LIN {X 0,Y 136.09,Z 552.523,A -85,B 0,C 180,E1 -24805.716,E2 -24805.716} C_VEL
LIN {X 0,Y 136.14,Z 552.524,A -85,B 0,C 180,E1 -24812.317,E2 -24812.317} C_VEL
LIN {X 0,Y 136.237,Z 552.49,A -85,B 0,C 180,E1 -24818.834,E2 -24818.834} C_VEL
LIN {X 0,Y 136.268,Z 552.51,A -85,B 0,C 180,E1 -24825.058,E2 -24825.058} C_VEL
LIN {X 0,Y 136.494,Z 552.467,A -85,B 0,C 180,E1 -24828.116,E2 -24828.116} C_VEL
LIN {X 0,Y 136.584,Z 552.444,A -85,B 0,C 180,E1 -24831.121,E2 -24831.121} C_VEL
LIN {X 0,Y 137.132,Z 552.379,A -85,B 0,C 180,E1 -24840.001,E2 -24840.001} C_VEL
LIN {X 0,Y 136.554,Z 552.471,A -85,B 0,C 180,E1 -24845.91,E2 -24845.91} C_VEL
LIN {X 0,Y 136.551,Z 552.458,A -85,B 0,C 180,E1 -24848.884,E2 -24848.884} C_VEL
LIN {X 0,Y 136.439,Z 552.483,A -85,B 0,C 180,E1 -24851.892,E2 -24851.892} C_VEL
LIN {X 0,Y 136.239,Z 552.503,A -85,B 0,C 180,E1 -24858.031,E2 -24858.031} C_VEL
LIN {X 0,Y 136.196,Z 552.518,A -85,B 0,C 180,E1 -24861.75,E2 -24861.75} C_VEL
LIN {X 0,Y 136.099,Z 552.528,A -85,B 0,C 180,E1 -24868.617,E2 -24868.617} C_VEL
LIN {X 0,Y 136.079,Z 552.53,A -85,B 0,C 180,E1 -24874.62,E2 -24874.62} C_VEL
LIN {X 0,Y 136.092,Z 552.641,A -85,B 0,C 180,E1 -24877.476,E2 -24877.476} C_VEL
LIN {X 0,Y 137.189,Z 555.484,A -85,B 0,C 180,E1 -24878.113,E2 -24878.113} C_VEL
LIN {X 0,Y 139.29,Z 558.883,A -85,B 0,C 180,E1 -24879.083,E2 -24879.083} C_VEL
LIN {X 0,Y 143.861,Z 567.914,A -85,B 0,C 180,E1 -24881.203,E2 -24881.203} C_VEL
LIN {X 0,Y 148.78,Z 578.743,A -85,B 0,C 180,E1 -24883.393,E2 -24883.393} C_VEL
LIN {X 0,Y 155.156,Z 595.109,A -85,B 0,C 180,E1 -24886.097,E2 -24886.097} C_VEL
LIN {X 0,Y 158.261,Z 604.425,A -85,B 0,C 180,E1 -24887.41,E2 -24887.41} C_VEL
LIN {X 0,Y 159.879,Z 625.259,A -85,B 0,C 180,E1 -24889.04,E2 -24889.04} C_VEL
LIN {X 0,Y 157.1,Z 663.701,A -85,B 0,C 180,E1 -24890.874,E2 -24890.874} C_VEL
LIN {X 0,Y 155.5,Z 676.27,A -85,B 0,C 180,E1 -24891.888,E2 -24891.888} C_VEL
LIN {X 0,Y 153.104,Z 689.007,A -85,B 0,C 180,E1 -24893.364,E2 -24893.364} C_VEL
LIN {X 0,Y 150.174,Z 701.556,A -85,B 0,C 180,E1 -24895.429,E2 -24895.429} C_VEL
LIN {X 0,Y 147.084,Z 712.81,A -85,B 0,C 180,E1 -24897.889,E2 -24897.889} C_VEL
LIN {X 0,Y 144.008,Z 723,A -85,B 0,C 180,E1 -24900.79,E2 -24900.79} C_VEL
LIN {X 0,Y 141.021,Z 732.187,A -85,B 0,C 180,E1 -24904.147,E2 -24904.147} C_VEL
LIN {X 0,Y 138.178,Z 741.159,A -85,B 0,C 180,E1 -24908.362,E2 -24908.362} C_VEL
LIN {X 0,Y 136.033,Z 748.303,A -85,B 0,C 180,E1 -24912.719,E2 -24912.719} C_VEL
LIN {X 0,Y 134.487,Z 754.79,A -85,B 0,C 180,E1 -24917.935,E2 -24917.935} C_VEL
LIN {X 0,Y 133.948,Z 759.008,A -85,B 0,C 180,E1 -24922.463,E2 -24922.463} C_VEL
LIN {X 0,Y 133.976,Z 762.099,A -85,B 0,C 180,E1 -24926.993,E2 -24926.993} C_VEL
LIN {X 0,Y 134.113,Z 763.587,A -85,B 0,C 180,E1 -24930,E2 -24930} C_VEL
LIN {X 0,Y 133.812,Z 764.716,A -85,B 0,C 180,E1 -24933.688,E2 -24933.688} C_VEL
LIN {X 0,Y 133.85,Z 765.305,A -85,B 0,C 180,E1 -24939.063,E2 -24939.063} C_VEL
LIN {X 0,Y 135.137,Z 764.541,A -85,B 0,C 180,E1 -24945.072,E2 -24945.072} C_VEL
LIN {X 0,Y 137.104,Z 762.867,A -85,B 0,C 180,E1 -24949.495,E2 -24949.495} C_VEL
LIN {X 0,Y 137.918,Z 761.696,A -85,B 0,C 180,E1 -24951.886,E2 -24951.886} C_VEL
LIN {X 0,Y 137.994,Z 759.344,A -85,B 0,C 180,E1 -24955.898,E2 -24955.898} C_VEL
LIN {X 0,Y 138.673,Z 756.379,A -85,B 0,C 180,E1 -24959.811,E2 -24959.811} C_VEL
LIN {X 0,Y 140.371,Z 754.198,A -85,B 0,C 180,E1 -24961.957,E2 -24961.957} C_VEL
LIN {X 0,Y 145.127,Z 749.46,A -85,B 0,C 180,E1 -24965.528,E2 -24965.528} C_VEL
LIN {X 0,Y 151.82,Z 742.178,A -85,B 0,C 180,E1 -24969.531,E2 -24969.531} C_VEL
LIN {X 0,Y 158.212,Z 734.316,A -85,B 0,C 180,E1 -24972.642,E2 -24972.642} C_VEL
LIN {X 0,Y 165.063,Z 724.645,A -85,B 0,C 180,E1 -24975.493,E2 -24975.493} C_VEL
LIN {X 0,Y 171.16,Z 714.802,A -85,B 0,C 180,E1 -24977.653,E2 -24977.653} C_VEL
LIN {X 0,Y 176.92,Z 703.823,A -85,B 0,C 180,E1 -24979.438,E2 -24979.438} C_VEL
LIN {X 0,Y 182.249,Z 691.549,A -85,B 0,C 180,E1 -24980.901,E2 -24980.901} C_VEL
LIN {X 0,Y 186.405,Z 679.587,A -85,B 0,C 180,E1 -24981.909,E2 -24981.909} C_VEL
LIN {X 0,Y 189.889,Z 665.627,A -85,B 0,C 180,E1 -24982.759,E2 -24982.759} C_VEL
LIN {X 0,Y 192.008,Z 652.096,A -85,B 0,C 180,E1 -24983.328,E2 -24983.328} C_VEL
LIN {X 0,Y 193.595,Z 637.242,A -85,B 0,C 180,E1 -24983.887,E2 -24983.887} C_VEL
LIN {X 0,Y 191.722,Z 630.79,A -85,B 0,C 180,E1 -24986.149,E2 -24986.149} C_VEL
LIN {X 0,Y 189.779,Z 625.016,A -85,B 0,C 180,E1 -24988.77,E2 -24988.77} C_VEL
LIN {X 0,Y 188.199,Z 620.471,A -85,B 0,C 180,E1 -24991.475,E2 -24991.475} C_VEL
LIN {X 0,Y 186.751,Z 616.287,A -85,B 0,C 180,E1 -24994.893,E2 -24994.893} C_VEL
LIN {X 0,Y 185.699,Z 613.263,A -85,B 0,C 180,E1 -25000.085,E2 -25000.085} C_VEL
LIN {X 0,Y 185.761,Z 613.151,A -85,B 0,C 180,E1 -25003.283,E2 -25003.283} C_VEL
LIN {X 0,Y 186.862,Z 614.042,A -85,B 0,C 180,E1 -25007.592,E2 -25007.592} C_VEL
LIN {X 0,Y 188.587,Z 617.563,A -85,B 0,C 180,E1 -25011.426,E2 -25011.426} C_VEL
LIN {X 0,Y 189.358,Z 618.568,A -85,B 0,C 180,E1 -25012.584,E2 -25012.584} C_VEL
LIN {X 0,Y 190.975,Z 622.294,A -85,B 0,C 180,E1 -25014.976,E2 -25014.976} C_VEL
LIN {X 0,Y 193.52,Z 627.528,A -85,B 0,C 180,E1 -25017.852,E2 -25017.852} C_VEL
LIN {X 0,Y 194.29,Z 629.917,A -85,B 0,C 180,E1 -25018.733,E2 -25018.733} C_VEL
LIN {X 0,Y 191.633,Z 651.966,A -85,B 0,C 180,E1 -25019.565,E2 -25019.565} C_VEL
LIN {X 0,Y 188.897,Z 665.523,A -85,B 0,C 180,E1 -25020.377,E2 -25020.377} C_VEL
LIN {X 0,Y 185.418,Z 677.774,A -85,B 0,C 180,E1 -25021.491,E2 -25021.491} C_VEL
LIN {X 0,Y 180.772,Z 690.105,A -85,B 0,C 180,E1 -25022.984,E2 -25022.984} C_VEL
LIN {X 0,Y 175.363,Z 701.546,A -85,B 0,C 180,E1 -25024.833,E2 -25024.833} C_VEL
LIN {X 0,Y 169.241,Z 712.199,A -85,B 0,C 180,E1 -25027.155,E2 -25027.155} C_VEL
LIN {X 0,Y 163.84,Z 720.173,A -85,B 0,C 180,E1 -25029.401,E2 -25029.401} C_VEL
LIN {X 0,Y 157.048,Z 728.925,A -85,B 0,C 180,E1 -25032.662,E2 -25032.662} C_VEL
LIN {X 0,Y 150.633,Z 735.958,A -85,B 0,C 180,E1 -25036.255,E2 -25036.255} C_VEL
LIN {X 0,Y 145.385,Z 741.003,A -85,B 0,C 180,E1 -25039.777,E2 -25039.777} C_VEL
LIN {X 0,Y 140.735,Z 744.941,A -85,B 0,C 180,E1 -25043.545,E2 -25043.545} C_VEL
LIN {X 0,Y 135.871,Z 748.426,A -85,B 0,C 180,E1 -25048.441,E2 -25048.441} C_VEL
LIN {X 0,Y 132.96,Z 750.107,A -85,B 0,C 180,E1 -25052.252,E2 -25052.252} C_VEL
LIN {X 0,Y 130.467,Z 751.138,A -85,B 0,C 180,E1 -25056.336,E2 -25056.336} C_VEL
LIN {X 0,Y 128.393,Z 751.409,A -85,B 0,C 180,E1 -25061.059,E2 -25061.059} C_VEL
LIN {X 0,Y 127.046,Z 750.731,A -85,B 0,C 180,E1 -25065.981,E2 -25065.981} C_VEL
LIN {X 0,Y 126.325,Z 748.479,A -85,B 0,C 180,E1 -25072.269,E2 -25072.269} C_VEL
LIN {X 0,Y 126.816,Z 744.824,A -85,B 0,C 180,E1 -25078.3,E2 -25078.3} C_VEL
LIN {X 0,Y 128.142,Z 739.779,A -85,B 0,C 180,E1 -25083.976,E2 -25083.976} C_VEL
LIN {X 0,Y 130.193,Z 733.128,A -85,B 0,C 180,E1 -25089.459,E2 -25089.459} C_VEL
LIN {X 0,Y 132.622,Z 725.996,A -85,B 0,C 180,E1 -25093.947,E2 -25093.947} C_VEL
LIN {X 0,Y 135.459,Z 717.663,A -85,B 0,C 180,E1 -25098.023,E2 -25098.023} C_VEL
LIN {X 0,Y 138.566,Z 708.298,A -85,B 0,C 180,E1 -25101.616,E2 -25101.616} C_VEL
LIN {X 0,Y 141.774,Z 697.812,A -85,B 0,C 180,E1 -25104.763,E2 -25104.763} C_VEL
LIN {X 0,Y 145.059,Z 685.612,A -85,B 0,C 180,E1 -25107.534,E2 -25107.534} C_VEL
LIN {X 0,Y 147.59,Z 674.21,A -85,B 0,C 180,E1 -25109.512,E2 -25109.512} C_VEL
LIN {X 0,Y 149.643,Z 662.69,A -85,B 0,C 180,E1 -25111.009,E2 -25111.009} C_VEL
LIN {X 0,Y 151.382,Z 648.86,A -85,B 0,C 180,E1 -25112.245,E2 -25112.245} C_VEL
LIN {X 0,Y 153.279,Z 624.867,A -85,B 0,C 180,E1 -25113.468,E2 -25113.468} C_VEL
LIN {X 0,Y 154.799,Z 601.404,A -85,B 0,C 180,E1 -25114.603,E2 -25114.603} C_VEL
LIN {X 0,Y 146.403,Z 582.461,A -85,B 0,C 180,E1 -25118.048,E2 -25118.048} C_VEL
LIN {X 0,Y 136.67,Z 565.458,A -85,B 0,C 180,E1 -25122.309,E2 -25122.309} C_VEL
LIN {X 0,Y 134.047,Z 561.533,A -85,B 0,C 180,E1 -25123.552,E2 -25123.552} C_VEL
LIN {X 0,Y 131.677,Z 557.899,A -85,B 0,C 180,E1 -25124.733,E2 -25124.733} C_VEL
LIN {X 0,Y 129.863,Z 555.601,A -85,B 0,C 180,E1 -25125.632,E2 -25125.632} C_VEL
LIN {X 0,Y 129.186,Z 553.389,A -85,B 0,C 180,E1 -25126.189,E2 -25126.189} C_VEL
LIN {X 0,Y 129.105,Z 553.398,A -85,B 0,C 180,E1 -25132.398,E2 -25132.398} C_VEL
LIN {X 0,Y 129.032,Z 553.409,A -85,B 0,C 180,E1 -25139.373,E2 -25139.373} C_VEL
LIN {X 0,Y 129.033,Z 553.412,A -85,B 0,C 180,E1 -25145.217,E2 -25145.217} C_VEL
LIN {X 0,Y 129.05,Z 553.4,A -85,B 0,C 180,E1 -25150.806,E2 -25150.806} C_VEL
LIN {X 0,Y 129.028,Z 553.407,A -85,B 0,C 180,E1 -25155.079,E2 -25155.079} C_VEL
LIN {X 0,Y 129.045,Z 553.395,A -85,B 0,C 180,E1 -25159.68,E2 -25159.68} C_VEL
LIN {X 0,Y 129.025,Z 553.406,A -85,B 0,C 180,E1 -25164.789,E2 -25164.789} C_VEL
LIN {X 0,Y 129.013,Z 553.404,A -85,B 0,C 180,E1 -25170.643,E2 -25170.643} C_VEL
LIN {X 0,Y 129.023,Z 553.413,A -85,B 0,C 180,E1 -25174.168,E2 -25174.168} C_VEL
LIN {X 0,Y 129.103,Z 553.383,A -85,B 0,C 180,E1 -25177.73,E2 -25177.73} C_VEL
LIN {X 0,Y 129.147,Z 553.378,A -85,B 0,C 180,E1 -25180.945,E2 -25180.945} C_VEL
LIN {X 0,Y 129.413,Z 553.351,A -85,B 0,C 180,E1 -25187.822,E2 -25187.822} C_VEL
LIN {X 0,Y 129.511,Z 553.323,A -85,B 0,C 180,E1 -25190.632,E2 -25190.632} C_VEL
LIN {X 0,Y 130.087,Z 553.255,A -85,B 0,C 180,E1 -25200.002,E2 -25200.002} C_VEL
LIN {X 0,Y 129.492,Z 553.35,A -85,B 0,C 180,E1 -25206.233,E2 -25206.233} C_VEL
LIN {X 0,Y 129.473,Z 553.338,A -85,B 0,C 180,E1 -25209.374,E2 -25209.374} C_VEL
LIN {X 0,Y 129.343,Z 553.37,A -85,B 0,C 180,E1 -25212.555,E2 -25212.555} C_VEL
LIN {X 0,Y 129.151,Z 553.39,A -85,B 0,C 180,E1 -25219.058,E2 -25219.058} C_VEL
LIN {X 0,Y 129.107,Z 553.399,A -85,B 0,C 180,E1 -25222.4,E2 -25222.4} C_VEL
LIN {X 0,Y 129.028,Z 553.409,A -85,B 0,C 180,E1 -25225.835,E2 -25225.835} C_VEL
LIN {X 0,Y 129.016,Z 553.408,A -85,B 0,C 180,E1 -25229.36,E2 -25229.36} C_VEL
LIN {X 0,Y 129.027,Z 553.409,A -85,B 0,C 180,E1 -25234.821,E2 -25234.821} C_VEL
LIN {X 0,Y 130.055,Z 556.296,A -85,B 0,C 180,E1 -25235.545,E2 -25235.545} C_VEL
LIN {X 0,Y 131.917,Z 558.677,A -85,B 0,C 180,E1 -25236.469,E2 -25236.469} C_VEL
LIN {X 0,Y 134.755,Z 563.668,A -85,B 0,C 180,E1 -25237.913,E2 -25237.913} C_VEL
LIN {X 0,Y 140.668,Z 575.654,A -85,B 0,C 180,E1 -25240.787,E2 -25240.787} C_VEL
LIN {X 0,Y 146.624,Z 590.149,A -85,B 0,C 180,E1 -25243.584,E2 -25243.584} C_VEL
LIN {X 0,Y 152.361,Z 606.452,A -85,B 0,C 180,E1 -25246.156,E2 -25246.156} C_VEL
LIN {X 0,Y 153.765,Z 625.671,A -85,B 0,C 180,E1 -25247.713,E2 -25247.713} C_VEL
LIN {X 0,Y 150.984,Z 663.049,A -85,B 0,C 180,E1 -25249.553,E2 -25249.553} C_VEL
LIN {X 0,Y 149.338,Z 675.367,A -85,B 0,C 180,E1 -25250.557,E2 -25250.557} C_VEL
LIN {X 0,Y 146.775,Z 688.765,A -85,B 0,C 180,E1 -25252.158,E2 -25252.158} C_VEL
LIN {X 0,Y 143.928,Z 700.467,A -85,B 0,C 180,E1 -25254.13,E2 -25254.13} C_VEL
LIN {X 0,Y 140.717,Z 711.834,A -85,B 0,C 180,E1 -25256.676,E2 -25256.676} C_VEL
LIN {X 0,Y 137.486,Z 722.143,A -85,B 0,C 180,E1 -25259.684,E2 -25259.684} C_VEL
LIN {X 0,Y 134.374,Z 731.375,A -85,B 0,C 180,E1 -25263.172,E2 -25263.172} C_VEL
LIN {X 0,Y 131.565,Z 739.736,A -85,B 0,C 180,E1 -25267.215,E2 -25267.215} C_VEL
LIN {X 0,Y 129.236,Z 747.093,A -85,B 0,C 180,E1 -25271.779,E2 -25271.779} C_VEL
LIN {X 0,Y 127.872,Z 752.035,A -85,B 0,C 180,E1 -25275.681,E2 -25275.681} C_VEL
LIN {X 0,Y 127.043,Z 756.812,A -85,B 0,C 180,E1 -25280.447,E2 -25280.447} C_VEL
LIN {X 0,Y 126.91,Z 760.54,A -85,B 0,C 180,E1 -25285.433,E2 -25285.433} C_VEL
LIN {X 0,Y 127.048,Z 762.903,A -85,B 0,C 180,E1 -25290,E2 -25290} C_VEL
LIN {X 0,Y 126.747,Z 764.071,A -85,B 0,C 180,E1 -25293.523,E2 -25293.523} C_VEL
LIN {X 0,Y 126.828,Z 764.858,A -85,B 0,C 180,E1 -25299.569,E2 -25299.569} C_VEL
LIN {X 0,Y 128.246,Z 764.222,A -85,B 0,C 180,E1 -25305.902,E2 -25305.902} C_VEL
LIN {X 0,Y 130.225,Z 762.838,A -85,B 0,C 180,E1 -25310.224,E2 -25310.224} C_VEL
LIN {X 0,Y 133.401,Z 760.406,A -85,B 0,C 180,E1 -25314.927,E2 -25314.927} C_VEL
LIN {X 0,Y 138.692,Z 755.849,A -85,B 0,C 180,E1 -25320.446,E2 -25320.446} C_VEL
LIN {X 0,Y 140.371,Z 754.198,A -85,B 0,C 180,E1 -25321.957,E2 -25321.957} C_VEL
LIN {X 0,Y 142.27,Z 751.869,A -85,B 0,C 180,E1 -25324.016,E2 -25324.016} C_VEL
LIN {X 0,Y 144.229,Z 747.781,A -85,B 0,C 180,E1 -25327.548,E2 -25327.548} C_VEL
LIN {X 0,Y 146.598,Z 743.171,A -85,B 0,C 180,E1 -25330.863,E2 -25330.863} C_VEL
LIN {X 0,Y 149.037,Z 739.974,A -85,B 0,C 180,E1 -25332.529,E2 -25332.529} C_VEL
LIN {X 0,Y 155.408,Z 732.316,A -85,B 0,C 180,E1 -25335.418,E2 -25335.418} C_VEL
LIN {X 0,Y 161.463,Z 724.147,A -85,B 0,C 180,E1 -25337.726,E2 -25337.726} C_VEL
LIN {X 0,Y 167.853,Z 714.275,A -85,B 0,C 180,E1 -25339.828,E2 -25339.828} C_VEL
LIN {X 0,Y 173.837,Z 703.262,A -85,B 0,C 180,E1 -25341.562,E2 -25341.562} C_VEL
LIN {X 0,Y 179.349,Z 690.955,A -85,B 0,C 180,E1 -25342.977,E2 -25342.977} C_VEL
LIN {X 0,Y 183.829,Z 678.287,A -85,B 0,C 180,E1 -25344.01,E2 -25344.01} C_VEL
LIN {X 0,Y 187.363,Z 664.446,A -85,B 0,C 180,E1 -25344.808,E2 -25344.808} C_VEL
LIN {X 0,Y 189.534,Z 650.679,A -85,B 0,C 180,E1 -25345.358,E2 -25345.358} C_VEL
LIN {X 0,Y 190.664,Z 640.493,A -85,B 0,C 180,E1 -25345.754,E2 -25345.754} C_VEL
LIN {X 0,Y 188.901,Z 634.168,A -85,B 0,C 180,E1 -25348.216,E2 -25348.216} C_VEL
LIN {X 0,Y 187.558,Z 629.89,A -85,B 0,C 180,E1 -25350.45,E2 -25350.45} C_VEL
LIN {X 0,Y 186.565,Z 626.764,A -85,B 0,C 180,E1 -25352.4,E2 -25352.4} C_VEL
LIN {X 0,Y 185.489,Z 623.054,A -85,B 0,C 180,E1 -25355.411,E2 -25355.411} C_VEL
LIN {X 0,Y 184.648,Z 620.365,A -85,B 0,C 180,E1 -25359.966,E2 -25359.966} C_VEL
LIN {X 0,Y 184.698,Z 620.152,A -85,B 0,C 180,E1 -25363.184,E2 -25363.184} C_VEL
LIN {X 0,Y 185.659,Z 621.005,A -85,B 0,C 180,E1 -25367.252,E2 -25367.252} C_VEL
LIN {X 0,Y 187.292,Z 624.444,A -85,B 0,C 180,E1 -25371.107,E2 -25371.107} C_VEL
LIN {X 0,Y 188.175,Z 625.92,A -85,B 0,C 180,E1 -25372.521,E2 -25372.521} C_VEL
LIN {X 0,Y 191.07,Z 632.698,A -85,B 0,C 180,E1 -25376.518,E2 -25376.518} C_VEL
LIN {X 0,Y 191.373,Z 633.441,A -85,B 0,C 180,E1 -25376.873,E2 -25376.873} C_VEL
LIN {X 0,Y 188.927,Z 652.714,A -85,B 0,C 180,E1 -25377.608,E2 -25377.608} C_VEL
LIN {X 0,Y 186.151,Z 665.828,A -85,B 0,C 180,E1 -25378.375,E2 -25378.375} C_VEL
LIN {X 0,Y 182.734,Z 677.45,A -85,B 0,C 180,E1 -25379.386,E2 -25379.386} C_VEL
LIN {X 0,Y 178.131,Z 689.355,A -85,B 0,C 180,E1 -25380.779,E2 -25380.779} C_VEL
LIN {X 0,Y 172.538,Z 700.982,A -85,B 0,C 180,E1 -25382.584,E2 -25382.584} C_VEL
LIN {X 0,Y 167.196,Z 710.185,A -85,B 0,C 180,E1 -25384.449,E2 -25384.449} C_VEL
LIN {X 0,Y 160.518,Z 719.842,A -85,B 0,C 180,E1 -25387.013,E2 -25387.013} C_VEL
LIN {X 0,Y 154.192,Z 727.701,A -85,B 0,C 180,E1 -25389.802,E2 -25389.802} C_VEL
LIN {X 0,Y 148.219,Z 734.146,A -85,B 0,C 180,E1 -25392.83,E2 -25392.83} C_VEL
LIN {X 0,Y 142.689,Z 739.381,A -85,B 0,C 180,E1 -25396.087,E2 -25396.087} C_VEL
LIN {X 0,Y 137.882,Z 743.427,A -85,B 0,C 180,E1 -25399.448,E2 -25399.448} C_VEL
LIN {X 0,Y 131.654,Z 747.895,A -85,B 0,C 180,E1 -25404.841,E2 -25404.841} C_VEL
LIN {X 0,Y 127.325,Z 750.317,A -85,B 0,C 180,E1 -25409.785,E2 -25409.785} C_VEL
LIN {X 0,Y 124.211,Z 751.537,A -85,B 0,C 180,E1 -25414.457,E2 -25414.457} C_VEL
LIN {X 0,Y 121.203,Z 751.74,A -85,B 0,C 180,E1 -25421.08,E2 -25421.08} C_VEL
LIN {X 0,Y 120.05,Z 751.064,A -85,B 0,C 180,E1 -25425.373,E2 -25425.373} C_VEL
LIN {X 0,Y 119.366,Z 749.619,A -85,B 0,C 180,E1 -25429.941,E2 -25429.941} C_VEL
LIN {X 0,Y 119.36,Z 746.867,A -85,B 0,C 180,E1 -25435.518,E2 -25435.518} C_VEL
LIN {X 0,Y 120.297,Z 742.793,A -85,B 0,C 180,E1 -25441.199,E2 -25441.199} C_VEL
LIN {X 0,Y 122.031,Z 736.887,A -85,B 0,C 180,E1 -25447.137,E2 -25447.137} C_VEL
LIN {X 0,Y 124.48,Z 729.689,A -85,B 0,C 180,E1 -25452.562,E2 -25452.562} C_VEL
LIN {X 0,Y 127.434,Z 721.432,A -85,B 0,C 180,E1 -25457.256,E2 -25457.256} C_VEL
LIN {X 0,Y 130.906,Z 711.723,A -85,B 0,C 180,E1 -25461.51,E2 -25461.51} C_VEL
LIN {X 0,Y 134.323,Z 701.288,A -85,B 0,C 180,E1 -25465.004,E2 -25465.004} C_VEL
LIN {X 0,Y 137.464,Z 690.498,A -85,B 0,C 180,E1 -25467.803,E2 -25467.803} C_VEL
LIN {X 0,Y 140.225,Z 679.539,A -85,B 0,C 180,E1 -25470,E2 -25470} C_VEL
LIN {X 0,Y 142.866,Z 666.494,A -85,B 0,C 180,E1 -25471.938,E2 -25471.938} C_VEL
LIN {X 0,Y 144.858,Z 652.649,A -85,B 0,C 180,E1 -25473.382,E2 -25473.382} C_VEL
LIN {X 0,Y 146.267,Z 637.699,A -85,B 0,C 180,E1 -25474.292,E2 -25474.292} C_VEL
LIN {X 0,Y 148.746,Z 603.405,A -85,B 0,C 180,E1 -25475.97,E2 -25475.97} C_VEL
LIN {X 0,Y 141.17,Z 586.11,A -85,B 0,C 180,E1 -25479.3,E2 -25479.3} C_VEL
LIN {X 0,Y 132.135,Z 570.127,A -85,B 0,C 180,E1 -25483.544,E2 -25483.544} C_VEL
LIN {X 0,Y 127.289,Z 562.863,A -85,B 0,C 180,E1 -25486.025,E2 -25486.025} C_VEL
LIN {X 0,Y 125.095,Z 559.496,A -85,B 0,C 180,E1 -25487.243,E2 -25487.243} C_VEL
LIN {X 0,Y 122.696,Z 556.329,A -85,B 0,C 180,E1 -25488.605,E2 -25488.605} C_VEL
LIN {X 0,Y 122.106,Z 554.27,A -85,B 0,C 180,E1 -25489.109,E2 -25489.109} C_VEL
LIN {X 0,Y 121.98,Z 554.288,A -85,B 0,C 180,E1 -25493.785,E2 -25493.785} C_VEL
LIN {X 0,Y 121.94,Z 554.293,A -85,B 0,C 180,E1 -25500.175,E2 -25500.175} C_VEL
LIN {X 0,Y 121.977,Z 554.289,A -85,B 0,C 180,E1 -25506.234,E2 -25506.234} C_VEL
LIN {X 0,Y 121.968,Z 554.286,A -85,B 0,C 180,E1 -25511.492,E2 -25511.492} C_VEL
LIN {X 0,Y 121.963,Z 554.27,A -85,B 0,C 180,E1 -25518.512,E2 -25518.512} C_VEL
LIN {X 0,Y 121.977,Z 554.284,A -85,B 0,C 180,E1 -25524.82,E2 -25524.82} C_VEL
LIN {X 0,Y 121.926,Z 554.278,A -85,B 0,C 180,E1 -25529.837,E2 -25529.837} C_VEL
LIN {X 0,Y 121.978,Z 554.281,A -85,B 0,C 180,E1 -25536.216,E2 -25536.216} C_VEL
LIN {X 0,Y 122.039,Z 554.257,A -85,B 0,C 180,E1 -25539.788,E2 -25539.788} C_VEL
LIN {X 0,Y 122.36,Z 554.231,A -85,B 0,C 180,E1 -25547.529,E2 -25547.529} C_VEL
LIN {X 0,Y 122.441,Z 554.203,A -85,B 0,C 180,E1 -25550.086,E2 -25550.086} C_VEL
LIN {X 0,Y 122.603,Z 554.206,A -85,B 0,C 180,E1 -25556.715,E2 -25556.715} C_VEL
LIN {X 0,Y 123.041,Z 554.132,A -85,B 0,C 180,E1 -25560.002,E2 -25560.002} C_VEL
LIN {X 0,Y 122.43,Z 554.228,A -85,B 0,C 180,E1 -25566.594,E2 -25566.594} C_VEL
LIN {X 0,Y 122.321,Z 554.244,A -85,B 0,C 180,E1 -25572.388,E2 -25572.388} C_VEL
LIN {X 0,Y 122.106,Z 554.262,A -85,B 0,C 180,E1 -25576.727,E2 -25576.727} C_VEL
LIN {X 0,Y 122.027,Z 554.277,A -85,B 0,C 180,E1 -25582.857,E2 -25582.857} C_VEL
LIN {X 0,Y 121.94,Z 554.297,A -85,B 0,C 180,E1 -25587.458,E2 -25587.458} C_VEL
LIN {X 0,Y 121.922,Z 554.32,A -85,B 0,C 180,E1 -25591.859,E2 -25591.859} C_VEL
LIN {X 0,Y 122.865,Z 557.041,A -85,B 0,C 180,E1 -25592.553,E2 -25592.553} C_VEL
LIN {X 0,Y 124.994,Z 559.604,A -85,B 0,C 180,E1 -25593.729,E2 -25593.729} C_VEL
LIN {X 0,Y 127.258,Z 563.09,A -85,B 0,C 180,E1 -25595.003,E2 -25595.003} C_VEL
LIN {X 0,Y 130.096,Z 568.017,A -85,B 0,C 180,E1 -25596.558,E2 -25596.558} C_VEL
LIN {X 0,Y 136.203,Z 580.763,A -85,B 0,C 180,E1 -25599.756,E2 -25599.756} C_VEL
LIN {X 0,Y 142.222,Z 596.004,A -85,B 0,C 180,E1 -25602.744,E2 -25602.744} C_VEL
LIN {X 0,Y 146.519,Z 608.877,A -85,B 0,C 180,E1 -25604.844,E2 -25604.844} C_VEL
LIN {X 0,Y 147.646,Z 627.078,A -85,B 0,C 180,E1 -25606.362,E2 -25606.362} C_VEL
LIN {X 0,Y 144.876,Z 662.586,A -85,B 0,C 180,E1 -25608.164,E2 -25608.164} C_VEL
LIN {X 0,Y 143.046,Z 675.642,A -85,B 0,C 180,E1 -25609.269,E2 -25609.269} C_VEL
LIN {X 0,Y 140.51,Z 688.326,A -85,B 0,C 180,E1 -25610.842,E2 -25610.842} C_VEL
LIN {X 0,Y 137.35,Z 700.828,A -85,B 0,C 180,E1 -25613.043,E2 -25613.043} C_VEL
LIN {X 0,Y 134,Z 712.051,A -85,B 0,C 180,E1 -25615.681,E2 -25615.681} C_VEL
LIN {X 0,Y 130.658,Z 722.22,A -85,B 0,C 180,E1 -25618.821,E2 -25618.821} C_VEL
LIN {X 0,Y 127.494,Z 731.235,A -85,B 0,C 180,E1 -25622.417,E2 -25622.417} C_VEL
LIN {X 0,Y 124.543,Z 739.665,A -85,B 0,C 180,E1 -25626.734,E2 -25626.734} C_VEL
LIN {X 0,Y 122.14,Z 746.958,A -85,B 0,C 180,E1 -25631.551,E2 -25631.551} C_VEL
LIN {X 0,Y 120.582,Z 752.736,A -85,B 0,C 180,E1 -25636.519,E2 -25636.519} C_VEL
LIN {X 0,Y 119.86,Z 757.241,A -85,B 0,C 180,E1 -25641.571,E2 -25641.571} C_VEL
LIN {X 0,Y 119.822,Z 760.6,A -85,B 0,C 180,E1 -25646.638,E2 -25646.638} C_VEL
LIN {X 0,Y 119.984,Z 762.218,A -85,B 0,C 180,E1 -25650,E2 -25650} C_VEL
LIN {X 0,Y 119.695,Z 763.37,A -85,B 0,C 180,E1 -25653.443,E2 -25653.443} C_VEL
LIN {X 0,Y 119.801,Z 764.407,A -85,B 0,C 180,E1 -25660.136,E2 -25660.136} C_VEL
LIN {X 0,Y 121.388,Z 763.902,A -85,B 0,C 180,E1 -25666.827,E2 -25666.827} C_VEL
LIN {X 0,Y 124.754,Z 761.933,A -85,B 0,C 180,E1 -25673.225,E2 -25673.225} C_VEL
LIN {X 0,Y 126.98,Z 760.364,A -85,B 0,C 180,E1 -25676.281,E2 -25676.281} C_VEL
LIN {X 0,Y 132.471,Z 756.078,A -85,B 0,C 180,E1 -25681.91,E2 -25681.91} C_VEL
LIN {X 0,Y 137.574,Z 751.551,A -85,B 0,C 180,E1 -25685.977,E2 -25685.977} C_VEL
LIN {X 0,Y 144.379,Z 744.971,A -85,B 0,C 180,E1 -25690.163,E2 -25690.163} C_VEL
LIN {X 0,Y 149.037,Z 739.974,A -85,B 0,C 180,E1 -25692.529,E2 -25692.529} C_VEL
LIN {X 0,Y 151.561,Z 736.607,A -85,B 0,C 180,E1 -25694.116,E2 -25694.116} C_VEL
LIN {X 0,Y 154.533,Z 730.969,A -85,B 0,C 180,E1 -25696.971,E2 -25696.971} C_VEL
LIN {X 0,Y 157.633,Z 724.825,A -85,B 0,C 180,E1 -25699.572,E2 -25699.572} C_VEL
LIN {X 0,Y 160.239,Z 720.669,A -85,B 0,C 180,E1 -25700.74,E2 -25700.74} C_VEL
LIN {X 0,Y 166.839,Z 710.406,A -85,B 0,C 180,E1 -25702.663,E2 -25702.663} C_VEL
LIN {X 0,Y 172.397,Z 700.122,A -85,B 0,C 180,E1 -25704.117,E2 -25704.117} C_VEL
LIN {X 0,Y 177.434,Z 688.881,A -85,B 0,C 180,E1 -25705.272,E2 -25705.272} C_VEL
LIN {X 0,Y 182.045,Z 675.604,A -85,B 0,C 180,E1 -25706.257,E2 -25706.257} C_VEL
LIN {X 0,Y 185.362,Z 662.219,A -85,B 0,C 180,E1 -25706.973,E2 -25706.973} C_VEL
LIN {X 0,Y 187.877,Z 645.028,A -85,B 0,C 180,E1 -25707.576,E2 -25707.576} C_VEL
LIN {X 0,Y 187.938,Z 643.927,A -85,B 0,C 180,E1 -25707.68,E2 -25707.68} C_VEL
LIN {X 0,Y 186.575,Z 638.505,A -85,B 0,C 180,E1 -25710.038,E2 -25710.038} C_VEL
LIN {X 0,Y 185.096,Z 633.268,A -85,B 0,C 180,E1 -25713.153,E2 -25713.153} C_VEL
LIN {X 0,Y 184.238,Z 629.822,A -85,B 0,C 180,E1 -25715.947,E2 -25715.947} C_VEL
LIN {X 0,Y 183.596,Z 627.486,A -85,B 0,C 180,E1 -25719.847,E2 -25719.847} C_VEL
LIN {X 0,Y 183.635,Z 627.166,A -85,B 0,C 180,E1 -25723.091,E2 -25723.091} C_VEL
LIN {X 0,Y 184.461,Z 627.981,A -85,B 0,C 180,E1 -25726.912,E2 -25726.912} C_VEL
LIN {X 0,Y 186,Z 631.347,A -85,B 0,C 180,E1 -25730.783,E2 -25730.783} C_VEL
LIN {X 0,Y 186.831,Z 633.123,A -85,B 0,C 180,E1 -25732.234,E2 -25732.234} C_VEL
LIN {X 0,Y 188.567,Z 637.673,A -85,B 0,C 180,E1 -25734.969,E2 -25734.969} C_VEL
LIN {X 0,Y 186.434,Z 653.605,A -85,B 0,C 180,E1 -25735.602,E2 -25735.602} C_VEL
LIN {X 0,Y 183.795,Z 665.679,A -85,B 0,C 180,E1 -25736.284,E2 -25736.284} C_VEL
LIN {X 0,Y 179.862,Z 678.546,A -85,B 0,C 180,E1 -25737.363,E2 -25737.363} C_VEL
LIN {X 0,Y 175.023,Z 690.496,A -85,B 0,C 180,E1 -25738.745,E2 -25738.745} C_VEL
LIN {X 0,Y 169.332,Z 701.751,A -85,B 0,C 180,E1 -25740.471,E2 -25740.471} C_VEL
LIN {X 0,Y 163.261,Z 711.575,A -85,B 0,C 180,E1 -25742.466,E2 -25742.466} C_VEL
LIN {X 0,Y 155.843,Z 721.607,A -85,B 0,C 180,E1 -25745.173,E2 -25745.173} C_VEL
LIN {X 0,Y 148.874,Z 729.649,A -85,B 0,C 180,E1 -25748.14,E2 -25748.14} C_VEL
LIN {X 0,Y 142.301,Z 736.131,A -85,B 0,C 180,E1 -25751.392,E2 -25751.392} C_VEL
LIN {X 0,Y 136.193,Z 741.344,A -85,B 0,C 180,E1 -25754.951,E2 -25754.951} C_VEL
LIN {X 0,Y 130.694,Z 745.42,A -85,B 0,C 180,E1 -25758.821,E2 -25758.821} C_VEL
LIN {X 0,Y 125.796,Z 748.515,A -85,B 0,C 180,E1 -25763.02,E2 -25763.02} C_VEL
LIN {X 0,Y 120.473,Z 751.12,A -85,B 0,C 180,E1 -25768.951,E2 -25768.951} C_VEL
LIN {X 0,Y 117.609,Z 752.045,A -85,B 0,C 180,E1 -25773.219,E2 -25773.219} C_VEL
LIN {X 0,Y 115.342,Z 752.294,A -85,B 0,C 180,E1 -25777.619,E2 -25777.619} C_VEL
LIN {X 0,Y 113.496,Z 751.745,A -85,B 0,C 180,E1 -25782.931,E2 -25782.931} C_VEL
LIN {X 0,Y 112.389,Z 750.207,A -85,B 0,C 180,E1 -25788.622,E2 -25788.622} C_VEL
LIN {X 0,Y 112.281,Z 746.882,A -85,B 0,C 180,E1 -25795.714,E2 -25795.714} C_VEL
LIN {X 0,Y 113.465,Z 742.005,A -85,B 0,C 180,E1 -25802.498,E2 -25802.498} C_VEL
LIN {X 0,Y 115.384,Z 735.975,A -85,B 0,C 180,E1 -25808.565,E2 -25808.565} C_VEL
LIN {X 0,Y 117.834,Z 729.025,A -85,B 0,C 180,E1 -25813.816,E2 -25813.816} C_VEL
LIN {X 0,Y 121.137,Z 720.322,A -85,B 0,C 180,E1 -25818.852,E2 -25818.852} C_VEL
LIN {X 0,Y 124.66,Z 710.638,A -85,B 0,C 180,E1 -25823.12,E2 -25823.12} C_VEL
LIN {X 0,Y 128.464,Z 699.456,A -85,B 0,C 180,E1 -25826.864,E2 -25826.864} C_VEL
LIN {X 0,Y 131.668,Z 688.694,A -85,B 0,C 180,E1 -25829.618,E2 -25829.618} C_VEL
LIN {X 0,Y 134.857,Z 675.993,A -85,B 0,C 180,E1 -25832.05,E2 -25832.05} C_VEL
LIN {X 0,Y 137.4,Z 663.097,A -85,B 0,C 180,E1 -25833.849,E2 -25833.849} C_VEL
LIN {X 0,Y 139.243,Z 649.243,A -85,B 0,C 180,E1 -25835.158,E2 -25835.158} C_VEL
LIN {X 0,Y 141.848,Z 618.247,A -85,B 0,C 180,E1 -25836.793,E2 -25836.793} C_VEL
LIN {X 0,Y 142.765,Z 605.565,A -85,B 0,C 180,E1 -25837.442,E2 -25837.442} C_VEL
LIN {X 0,Y 136.173,Z 590.148,A -85,B 0,C 180,E1 -25840.544,E2 -25840.544} C_VEL
LIN {X 0,Y 127.507,Z 574.615,A -85,B 0,C 180,E1 -25844.906,E2 -25844.906} C_VEL
LIN {X 0,Y 122.866,Z 567.639,A -85,B 0,C 180,E1 -25847.454,E2 -25847.454} C_VEL
LIN {X 0,Y 120.218,Z 563.637,A -85,B 0,C 180,E1 -25849.051,E2 -25849.051} C_VEL
LIN {X 0,Y 118.32,Z 560.661,A -85,B 0,C 180,E1 -25850.266,E2 -25850.266} C_VEL
LIN {X 0,Y 117.266,Z 559.549,A -85,B 0,C 180,E1 -25850.907,E2 -25850.907} C_VEL
LIN {X 0,Y 115.501,Z 557.134,A -85,B 0,C 180,E1 -25852.079,E2 -25852.079} C_VEL
LIN {X 0,Y 114.991,Z 555.156,A -85,B 0,C 180,E1 -25852.649,E2 -25852.649} C_VEL
LIN {X 0,Y 114.868,Z 555.177,A -85,B 0,C 180,E1 -25861.07,E2 -25861.07} C_VEL
LIN {X 0,Y 114.891,Z 555.16,A -85,B 0,C 180,E1 -25867.712,E2 -25867.712} C_VEL
LIN {X 0,Y 114.882,Z 555.173,A -85,B 0,C 180,E1 -25872.771,E2 -25872.771} C_VEL
LIN {X 0,Y 114.886,Z 555.151,A -85,B 0,C 180,E1 -25877.71,E2 -25877.71} C_VEL
LIN {X 0,Y 114.891,Z 555.172,A -85,B 0,C 180,E1 -25882.674,E2 -25882.674} C_VEL
LIN {X 0,Y 114.861,Z 555.152,A -85,B 0,C 180,E1 -25888.937,E2 -25888.937} C_VEL
LIN {X 0,Y 114.943,Z 555.154,A -85,B 0,C 180,E1 -25896.51,E2 -25896.51} C_VEL
LIN {X 0,Y 115.007,Z 555.147,A -85,B 0,C 180,E1 -25902.211,E2 -25902.211} C_VEL
LIN {X 0,Y 115.281,Z 555.114,A -85,B 0,C 180,E1 -25907.265,E2 -25907.265} C_VEL
LIN {X 0,Y 115.384,Z 555.097,A -85,B 0,C 180,E1 -25913.005,E2 -25913.005} C_VEL
LIN {X 0,Y 115.993,Z 555.009,A -85,B 0,C 180,E1 -25920.002,E2 -25920.002} C_VEL
LIN {X 0,Y 115.369,Z 555.105,A -85,B 0,C 180,E1 -25927,E2 -25927} C_VEL
LIN {X 0,Y 115.254,Z 555.125,A -85,B 0,C 180,E1 -25932.675,E2 -25932.675} C_VEL
LIN {X 0,Y 115.009,Z 555.145,A -85,B 0,C 180,E1 -25937.792,E2 -25937.792} C_VEL
LIN {X 0,Y 114.947,Z 555.156,A -85,B 0,C 180,E1 -25943.494,E2 -25943.494} C_VEL
LIN {X 0,Y 114.883,Z 555.232,A -85,B 0,C 180,E1 -25948.428,E2 -25948.428} C_VEL
LIN {X 0,Y 115.821,Z 557.945,A -85,B 0,C 180,E1 -25949.221,E2 -25949.221} C_VEL
LIN {X 0,Y 118.137,Z 560.716,A -85,B 0,C 180,E1 -25950.686,E2 -25950.686} C_VEL
LIN {X 0,Y 120.216,Z 563.917,A -85,B 0,C 180,E1 -25951.994,E2 -25951.994} C_VEL
LIN {X 0,Y 121.3,Z 565.531,A -85,B 0,C 180,E1 -25952.655,E2 -25952.655} C_VEL
LIN {X 0,Y 125.165,Z 571.603,A -85,B 0,C 180,E1 -25954.894,E2 -25954.894} C_VEL
LIN {X 0,Y 131.123,Z 584.399,A -85,B 0,C 180,E1 -25958.299,E2 -25958.299} C_VEL
LIN {X 0,Y 136.997,Z 599.716,A -85,B 0,C 180,E1 -25961.462,E2 -25961.462} C_VEL
LIN {X 0,Y 140.721,Z 610.697,A -85,B 0,C 180,E1 -25963.373,E2 -25963.373} C_VEL
LIN {X 0,Y 141.716,Z 626.93,A -85,B 0,C 180,E1 -25964.819,E2 -25964.819} C_VEL
LIN {X 0,Y 138.854,Z 662.115,A -85,B 0,C 180,E1 -25966.651,E2 -25966.651} C_VEL
LIN {X 0,Y 137.113,Z 674.49,A -85,B 0,C 180,E1 -25967.722,E2 -25967.722} C_VEL
LIN {X 0,Y 134.319,Z 687.883,A -85,B 0,C 180,E1 -25969.402,E2 -25969.402} C_VEL
LIN {X 0,Y 131.266,Z 699.613,A -85,B 0,C 180,E1 -25971.509,E2 -25971.509} C_VEL
LIN {X 0,Y 127.771,Z 710.987,A -85,B 0,C 180,E1 -25974.239,E2 -25974.239} C_VEL
LIN {X 0,Y 124.231,Z 721.297,A -85,B 0,C 180,E1 -25977.492,E2 -25977.492} C_VEL
LIN {X 0,Y 120.642,Z 731.061,A -85,B 0,C 180,E1 -25981.565,E2 -25981.565} C_VEL
LIN {X 0,Y 117.513,Z 739.571,A -85,B 0,C 180,E1 -25986.191,E2 -25986.191} C_VEL
LIN {X 0,Y 115.033,Z 746.785,A -85,B 0,C 180,E1 -25991.292,E2 -25991.292} C_VEL
LIN {X 0,Y 113.648,Z 751.635,A -85,B 0,C 180,E1 -25995.679,E2 -25995.679} C_VEL
LIN {X 0,Y 112.84,Z 756.305,A -85,B 0,C 180,E1 -26001.042,E2 -26001.042} C_VEL
LIN {X 0,Y 112.759,Z 759.796,A -85,B 0,C 180,E1 -26006.427,E2 -26006.427} C_VEL
LIN {X 0,Y 112.92,Z 761.508,A -85,B 0,C 180,E1 -26010,E2 -26010} C_VEL
LIN {X 0,Y 112.626,Z 762.702,A -85,B 0,C 180,E1 -26013.578,E2 -26013.578} C_VEL
LIN {X 0,Y 112.802,Z 763.911,A -85,B 0,C 180,E1 -26020.772,E2 -26020.772} C_VEL
LIN {X 0,Y 113.486,Z 763.95,A -85,B 0,C 180,E1 -26024.342,E2 -26024.342} C_VEL
LIN {X 0,Y 116.18,Z 762.858,A -85,B 0,C 180,E1 -26031.281,E2 -26031.281} C_VEL
LIN {X 0,Y 120.642,Z 760.3,A -85,B 0,C 180,E1 -26037.777,E2 -26037.777} C_VEL
LIN {X 0,Y 126.105,Z 756.514,A -85,B 0,C 180,E1 -26043.281,E2 -26043.281} C_VEL
LIN {X 0,Y 131.907,Z 751.863,A -85,B 0,C 180,E1 -26047.785,E2 -26047.785} C_VEL
LIN {X 0,Y 139.048,Z 745.511,A -85,B 0,C 180,E1 -26052.043,E2 -26052.043} C_VEL
LIN {X 0,Y 145.778,Z 738.697,A -85,B 0,C 180,E1 -26055.323,E2 -26055.323} C_VEL
LIN {X 0,Y 153.044,Z 730.336,A -85,B 0,C 180,E1 -26058.263,E2 -26058.263} C_VEL
LIN {X 0,Y 160.239,Z 720.669,A -85,B 0,C 180,E1 -26060.74,E2 -26060.74} C_VEL
LIN {X 0,Y 161.875,Z 717.847,A -85,B 0,C 180,E1 -26061.553,E2 -26061.553} C_VEL
LIN {X 0,Y 165.055,Z 708.967,A -85,B 0,C 180,E1 -26064.946,E2 -26064.946} C_VEL
LIN {X 0,Y 166.611,Z 705.818,A -85,B 0,C 180,E1 -26065.606,E2 -26065.606} C_VEL
LIN {X 0,Y 172.792,Z 693.744,A -85,B 0,C 180,E1 -26067.02,E2 -26067.02} C_VEL
LIN {X 0,Y 178.041,Z 680.765,A -85,B 0,C 180,E1 -26068.052,E2 -26068.052} C_VEL
LIN {X 0,Y 182.051,Z 667.402,A -85,B 0,C 180,E1 -26068.84,E2 -26068.84} C_VEL
LIN {X 0,Y 184.756,Z 653.544,A -85,B 0,C 180,E1 -26069.395,E2 -26069.395} C_VEL
LIN {X 0,Y 185.528,Z 647.693,A -85,B 0,C 180,E1 -26069.603,E2 -26069.603} C_VEL
LIN {X 0,Y 184.375,Z 642.729,A -85,B 0,C 180,E1 -26072.044,E2 -26072.044} C_VEL
LIN {X 0,Y 183.619,Z 639.517,A -85,B 0,C 180,E1 -26074.123,E2 -26074.123} C_VEL
LIN {X 0,Y 182.917,Z 636.385,A -85,B 0,C 180,E1 -26076.806,E2 -26076.806} C_VEL
LIN {X 0,Y 182.487,Z 634.265,A -85,B 0,C 180,E1 -26080.834,E2 -26080.834} C_VEL
LIN {X 0,Y 182.999,Z 634.547,A -85,B 0,C 180,E1 -26085.507,E2 -26085.507} C_VEL
LIN {X 0,Y 183.303,Z 635.076,A -85,B 0,C 180,E1 -26086.699,E2 -26086.699} C_VEL
LIN {X 0,Y 185.004,Z 638.852,A -85,B 0,C 180,E1 -26090.995,E2 -26090.995} C_VEL
LIN {X 0,Y 186.106,Z 642.095,A -85,B 0,C 180,E1 -26093.029,E2 -26093.029} C_VEL
LIN {X 0,Y 184.117,Z 655.476,A -85,B 0,C 180,E1 -26093.585,E2 -26093.585} C_VEL
LIN {X 0,Y 181.129,Z 667.979,A -85,B 0,C 180,E1 -26094.292,E2 -26094.292} C_VEL
LIN {X 0,Y 177.007,Z 680.362,A -85,B 0,C 180,E1 -26095.354,E2 -26095.354} C_VEL
LIN {X 0,Y 172.178,Z 691.591,A -85,B 0,C 180,E1 -26096.639,E2 -26096.639} C_VEL
LIN {X 0,Y 166.1,Z 702.995,A -85,B 0,C 180,E1 -26098.364,E2 -26098.364} C_VEL
LIN {X 0,Y 159.927,Z 712.494,A -85,B 0,C 180,E1 -26100.258,E2 -26100.258} C_VEL
LIN {X 0,Y 152.956,Z 721.533,A -85,B 0,C 180,E1 -26102.632,E2 -26102.632} C_VEL
LIN {X 0,Y 145.571,Z 729.688,A -85,B 0,C 180,E1 -26105.54,E2 -26105.54} C_VEL
LIN {X 0,Y 138.563,Z 736.253,A -85,B 0,C 180,E1 -26108.751,E2 -26108.751} C_VEL
LIN {X 0,Y 132.032,Z 741.546,A -85,B 0,C 180,E1 -26112.292,E2 -26112.292} C_VEL
LIN {X 0,Y 124.946,Z 746.397,A -85,B 0,C 180,E1 -26117.021,E2 -26117.021} C_VEL
LIN {X 0,Y 120.296,Z 749.048,A -85,B 0,C 180,E1 -26120.814,E2 -26120.814} C_VEL
LIN {X 0,Y 116.088,Z 751.025,A -85,B 0,C 180,E1 -26125.072,E2 -26125.072} C_VEL
LIN {X 0,Y 112.202,Z 752.312,A -85,B 0,C 180,E1 -26130.071,E2 -26130.071} C_VEL
LIN {X 0,Y 109.048,Z 752.734,A -85,B 0,C 180,E1 -26135.451,E2 -26135.451} C_VEL
LIN {X 0,Y 106.833,Z 752.242,A -85,B 0,C 180,E1 -26141.134,E2 -26141.134} C_VEL
LIN {X 0,Y 105.344,Z 750.445,A -85,B 0,C 180,E1 -26148.154,E2 -26148.154} C_VEL
LIN {X 0,Y 105.179,Z 747.048,A -85,B 0,C 180,E1 -26155.599,E2 -26155.599} C_VEL
LIN {X 0,Y 106.284,Z 742.424,A -85,B 0,C 180,E1 -26162.428,E2 -26162.428} C_VEL
LIN {X 0,Y 107.935,Z 737.308,A -85,B 0,C 180,E1 -26168.013,E2 -26168.013} C_VEL
LIN {X 0,Y 110.147,Z 731.262,A -85,B 0,C 180,E1 -26173.146,E2 -26173.146} C_VEL
LIN {X 0,Y 113.276,Z 723.309,A -85,B 0,C 180,E1 -26178.367,E2 -26178.367} C_VEL
LIN {X 0,Y 116.957,Z 713.825,A -85,B 0,C 180,E1 -26183.098,E2 -26183.098} C_VEL
LIN {X 0,Y 120.786,Z 703.353,A -85,B 0,C 180,E1 -26187.082,E2 -26187.082} C_VEL
LIN {X 0,Y 124.409,Z 692.186,A -85,B 0,C 180,E1 -26190.282,E2 -26190.282} C_VEL
LIN {X 0,Y 127.732,Z 680.305,A -85,B 0,C 180,E1 -26192.86,E2 -26192.86} C_VEL
LIN {X 0,Y 130.476,Z 667.998,A -85,B 0,C 180,E1 -26194.828,E2 -26194.828} C_VEL
LIN {X 0,Y 132.641,Z 654.532,A -85,B 0,C 180,E1 -26196.351,E2 -26196.351} C_VEL
LIN {X 0,Y 134.136,Z 640.934,A -85,B 0,C 180,E1 -26197.29,E2 -26197.29} C_VEL
LIN {X 0,Y 136.822,Z 607.674,A -85,B 0,C 180,E1 -26198.997,E2 -26198.997} C_VEL
LIN {X 0,Y 131.367,Z 594.491,A -85,B 0,C 180,E1 -26201.814,E2 -26201.814} C_VEL
LIN {X 0,Y 122.905,Z 578.995,A -85,B 0,C 180,E1 -26206.379,E2 -26206.379} C_VEL
LIN {X 0,Y 116.329,Z 568.921,A -85,B 0,C 180,E1 -26210.414,E2 -26210.414} C_VEL
LIN {X 0,Y 113.896,Z 565.384,A -85,B 0,C 180,E1 -26212.044,E2 -26212.044} C_VEL
LIN {X 0,Y 111.615,Z 562.183,A -85,B 0,C 180,E1 -26213.667,E2 -26213.667} C_VEL
LIN {X 0,Y 110.827,Z 560.96,A -85,B 0,C 180,E1 -26214.271,E2 -26214.271} C_VEL
LIN {X 0,Y 108.722,Z 558.774,A -85,B 0,C 180,E1 -26215.833,E2 -26215.833} C_VEL
LIN {X 0,Y 107.785,Z 556.055,A -85,B 0,C 180,E1 -26216.952,E2 -26216.952} C_VEL
LIN {X 0,Y 107.8,Z 556.056,A -85,B 0,C 180,E1 -26222.059,E2 -26222.059} C_VEL
LIN {X 0,Y 107.791,Z 556.04,A -85,B 0,C 180,E1 -26228.522,E2 -26228.522} C_VEL
LIN {X 0,Y 107.781,Z 556.045,A -85,B 0,C 180,E1 -26235.828,E2 -26235.828} C_VEL
LIN {X 0,Y 107.786,Z 556.053,A -85,B 0,C 180,E1 -26241.483,E2 -26241.483} C_VEL
LIN {X 0,Y 107.804,Z 556.029,A -85,B 0,C 180,E1 -26248.567,E2 -26248.567} C_VEL
LIN {X 0,Y 107.907,Z 556.025,A -85,B 0,C 180,E1 -26256.999,E2 -26256.999} C_VEL
LIN {X 0,Y 108.033,Z 556.026,A -85,B 0,C 180,E1 -26264.919,E2 -26264.919} C_VEL
LIN {X 0,Y 108.284,Z 555.97,A -85,B 0,C 180,E1 -26268.774,E2 -26268.774} C_VEL
LIN {X 0,Y 108.454,Z 555.969,A -85,B 0,C 180,E1 -26276.286,E2 -26276.286} C_VEL
LIN {X 0,Y 108.943,Z 555.887,A -85,B 0,C 180,E1 -26280.002,E2 -26280.002} C_VEL
LIN {X 0,Y 108.307,Z 555.981,A -85,B 0,C 180,E1 -26287.459,E2 -26287.459} C_VEL
